DATA_BLOCK "SP201"   // DB235
// stored: MemoryReserve 100
   VAR
      "MAIN OP AUTO INITIATE PBL (GREEN)" : Bool := FALSE;
      "MAIN OP STOP PBL (RED)" : Bool := FALSE;
      RESERVE : Bool := FALSE;
      SPARE : Bool := FALSE;
      SPARE_1 : Bool := FALSE;
      SPARE_2 : Bool := FALSE;
      SPARE_3 : Bool := FALSE;
      SPARE_4 : Bool := FALSE;
      "MAIN HMI POWER TRIPPED E110CB" : Bool := TRUE;
   END_VAR
BEGIN
END_DATA_BLOCK

DATA_BLOCK "SP202"   // DB345
// stored: MemoryReserve 100
   VAR
      "AUTO INITIATE PBL LAMP (GREEN)" : Bool := FALSE;
      "STOP PBL LAMP ON (RED)" : Bool := TRUE;
      SPARE_4 : Bool := FALSE;
      "ENABLE PBL LAMP ON (BLACK)" : Bool := FALSE;
      "SAFETY RESET PBL LAMP (BLUE)" : Bool := FALSE;
      SPARE : Bool := FALSE;
      SPARE_1 : Bool := FALSE;
      SPARE_2 : Bool := FALSE;
      "TOWER LAMP 1 ON (RED)" : Bool := TRUE;
      "TOWER LAMP 2 ON (AMBER)" : Bool := FALSE;
      "TOWER LAMP 3 ON (GREEN)" : Bool := FALSE;
      "TOWER LAMP 4 ON (WHITE)" : Bool := FALSE;
      "TOWER LAMP 5 ON (BLUE)" : Bool := FALSE;
      "Buzzer On" : Bool := FALSE;
      SPARE_3 : Bool := FALSE;
      SPARE_5 : Bool := FALSE;
   END_VAR
BEGIN
END_DATA_BLOCK

DATA_BLOCK "SP203"   // DB346
// stored: MemoryReserve 100
   VAR
      "MODE SELECT AUTO" : Bool := FALSE;
      "HOME PBL (GREEN)" : Bool := FALSE;
      "SAFETY RESET PBL (BLUE)" : Bool := FALSE;
      "SCS MODE SELECT AUTO" : Bool := FALSE;
      "MODE SELECT MANUAL" : Bool := TRUE;
      "ENABLE PBL (BLACK)" : Bool := FALSE;
      "SCS MODE SELECT SETUP" : Bool := TRUE;
      "SCS MODE SELECT DISABLE" : Bool := FALSE;
   END_VAR
BEGIN
END_DATA_BLOCK

DATA_BLOCK "SP204"   // DB344
// stored: MemoryReserve 100
   VAR
      "MAIN OP EMERGENCY STOP CH.A" : Bool := TRUE;
      SPARE : Bool := FALSE;
      SPARE_1 : Bool := FALSE;
      SPARE_2 : Bool := FALSE;
      "MAIN OP EMERGENCY STOP CH.B" : Bool := FALSE;
   END_VAR
BEGIN
END_DATA_BLOCK

DATA_BLOCK "SP205"   // DB343
// stored: MemoryReserve 100
   VAR
      "PENDANT REQUIRED PL (YELLOW)" : Bool := TRUE;
      SPARE : Bool := FALSE;
      "HOME PBL LAMP ON (GREEN)" : Bool := FALSE;
      SPARE_1 : Bool := FALSE;
      SPARE_2 : Bool := FALSE;
      SPARE_3 : Bool := FALSE;
      SPARE_4 : Bool := FALSE;
      "SCS SELECT DISABLE PL (GREEN)" : Bool := TRUE;
   END_VAR
BEGIN
END_DATA_BLOCK

DATA_BLOCK "SP501"   // DB341
// stored: MemoryReserve 100
   VAR
      "CONTROL DC POWER TRIPPED E156CB" : Bool := TRUE;
      "SAFETY DC POWER TRIPPED E218CB" : Bool := TRUE;
      "CLASS 2 SMPS POWER TRIPPED E308CB" : Bool := TRUE;
      "CLASS 2 SMPS MONITORING E310PWS" : Bool := TRUE;
      "ET200ECO PN-1 POWER TRIPPED E324CB" : Bool := TRUE;
      "ET200ECO PN-2 POWER TRIPPED E328CB" : Bool := TRUE;
      "ET200ECO PN-3 POWER TRIPPED E332CB" : Bool := TRUE;
      "ET200ECO PN-4 POWER TRIPPED E336CB" : Bool := TRUE;
      "SEPA UW IONIZER TOP MAINTERNANCE DETECTION" : Bool := FALSE;
      "SEPA UW IONIZER TOP ERROR" : Bool := TRUE;
      SPARE : Bool := FALSE;
      SPARE_1 : Bool := FALSE;
      "SEPA UW IONIZER BOTTOM MAINTERNANCE DETECTION" : Bool := FALSE;
      "SEPA UW IONIZER BOTTOM ERROR" : Bool := TRUE;
      SPARE_2 : Bool := FALSE;
      SPARE_3 : Bool := FALSE;
   END_VAR
BEGIN
END_DATA_BLOCK

DATA_BLOCK "SP502"   // DB340
// stored: MemoryReserve 100
   VAR
      "CLASS2 SMPS ALARM RESET" : Bool := FALSE;
      SPARE_4 : Bool := FALSE;
      SPARE_5 : Bool := FALSE;
      SPARE_6 : Bool := FALSE;
      SPARE_7 : Bool := FALSE;
      SPARE_8 : Bool := FALSE;
      SPARE_9 : Bool := FALSE;
      SPARE_10 : Bool := FALSE;
      "SEPA UW IONIZER TOP MAINTERNANCE DETECTION" : Bool := FALSE;
      "SEPA UW IONIZER TOP DISCHARGE STOP" : Bool := FALSE;
      SPARE : Bool := FALSE;
      SPARE_1 : Bool := FALSE;
      "SEPA UW IONIZER BOTTOM MAINTERNANCE DETECTION" : Bool := FALSE;
      "SEPA UW IONIZER BOTTOM DISCHARGE STOP" : Bool := FALSE;
   END_VAR
BEGIN
END_DATA_BLOCK

DATA_BLOCK "SP506"   // DB234
// stored: MemoryReserve 100
   VAR
      "PHMI EMERGENCY STOP CH.A" : Bool := TRUE;
      "PHMI ENABLE SWITCH CH.A" : Bool := FALSE;
      SPARE : Bool := FALSE;
      SPARE_1 : Bool := FALSE;
      "PHMI EMERGENCY STOP CH.B" : Bool := FALSE;
      "PHMI ENABLE SWITCH CH.B" : Bool := FALSE;
   END_VAR
BEGIN
END_DATA_BLOCK

DATA_BLOCK "SP507"   // DB339
// stored: MemoryReserve 100
   VAR
      "UNWINDER EPCC01 INTERLOCK" : Bool := FALSE;
      "UNWINDER EPCC02 INTERLOCK" : Bool := FALSE;
      "UNWINDER EPCC03 INTERLOCK" : Bool := FALSE;
      "UNWINDER EPCC04 INTERLOCK" : Bool := FALSE;
   END_VAR
BEGIN
END_DATA_BLOCK

DATA_BLOCK "SP508"   // DB342
// stored: MemoryReserve 100
   VAR
      "ANODE ALIGN VISION BUSY (STO)" : Bool := FALSE;
      "ANODE ALIGN VISION RESULT (OK)" : Bool := TRUE;
      "STACK VISION BUSY (STO)" : Bool := FALSE;
      "STACK VISION RESULT (OK)" : Bool := FALSE;
      "CATHODE ALIGN VISION BUSY (STO)" : Bool := FALSE;
      "CATHODE ALIGN VISION RESULT (OK)" : Bool := FALSE;
   END_VAR
BEGIN
END_DATA_BLOCK

DATA_BLOCK "IdentRfHmi"   // DB213
// stored: MemoryReserve 100
   VAR
      unitIdentRf : Array[0.."NO_OF_UNITS"] of "typeEMIdentRf";
   END_VAR
BEGIN
   unitIdentRf[0].identRfEM[0..7].selectedUnit := 0;
   unitIdentRf[0].identRfEM[0..7].selectedEM := 0;
   unitIdentRf[0].identRfEM[0..7].rfReaderId := 0;
   unitIdentRf[0].identRfEM[0..7].numberOfRf := 0;
   unitIdentRf[0].identRfEM[0].rfReader[0..1].deviceName := WSTRING#'';
   unitIdentRf[0].identRfEM[1].rfReader[0..1].deviceName := WSTRING#'';
   unitIdentRf[0].identRfEM[2].rfReader[0..1].deviceName := WSTRING#'';
   unitIdentRf[0].identRfEM[3].rfReader[0..1].deviceName := WSTRING#'';
   unitIdentRf[0].identRfEM[4].rfReader[0..1].deviceName := WSTRING#'';
   unitIdentRf[0].identRfEM[5].rfReader[0..1].deviceName := WSTRING#'';
   unitIdentRf[0].identRfEM[6].rfReader[0..1].deviceName := WSTRING#'';
   unitIdentRf[0].identRfEM[7].rfReader[0..1].deviceName := WSTRING#'';
   unitIdentRf[0].identRfEM[0].rfReader[0..1].deviceType := WSTRING#'';
   unitIdentRf[0].identRfEM[1].rfReader[0..1].deviceType := WSTRING#'';
   unitIdentRf[0].identRfEM[2].rfReader[0..1].deviceType := WSTRING#'';
   unitIdentRf[0].identRfEM[3].rfReader[0..1].deviceType := WSTRING#'';
   unitIdentRf[0].identRfEM[4].rfReader[0..1].deviceType := WSTRING#'';
   unitIdentRf[0].identRfEM[5].rfReader[0..1].deviceType := WSTRING#'';
   unitIdentRf[0].identRfEM[6].rfReader[0..1].deviceType := WSTRING#'';
   unitIdentRf[0].identRfEM[7].rfReader[0..1].deviceType := WSTRING#'';
   unitIdentRf[0].identRfEM[0].rfReader[0..1].deviceId := 0;
   unitIdentRf[0].identRfEM[1].rfReader[0..1].deviceId := 0;
   unitIdentRf[0].identRfEM[2].rfReader[0..1].deviceId := 0;
   unitIdentRf[0].identRfEM[3].rfReader[0..1].deviceId := 0;
   unitIdentRf[0].identRfEM[4].rfReader[0..1].deviceId := 0;
   unitIdentRf[0].identRfEM[5].rfReader[0..1].deviceId := 0;
   unitIdentRf[0].identRfEM[6].rfReader[0..1].deviceId := 0;
   unitIdentRf[0].identRfEM[7].rfReader[0..1].deviceId := 0;
   unitIdentRf[0].identRfEM[0].rfReader[0..1].tagType := WSTRING#'';
   unitIdentRf[0].identRfEM[1].rfReader[0..1].tagType := WSTRING#'';
   unitIdentRf[0].identRfEM[2].rfReader[0..1].tagType := WSTRING#'';
   unitIdentRf[0].identRfEM[3].rfReader[0..1].tagType := WSTRING#'';
   unitIdentRf[0].identRfEM[4].rfReader[0..1].tagType := WSTRING#'';
   unitIdentRf[0].identRfEM[5].rfReader[0..1].tagType := WSTRING#'';
   unitIdentRf[0].identRfEM[6].rfReader[0..1].tagType := WSTRING#'';
   unitIdentRf[0].identRfEM[7].rfReader[0..1].tagType := WSTRING#'';
   unitIdentRf[0].identRfEM[0].rfReader[0..1].cameraMode := WSTRING#'';
   unitIdentRf[0].identRfEM[1].rfReader[0..1].cameraMode := WSTRING#'';
   unitIdentRf[0].identRfEM[2].rfReader[0..1].cameraMode := WSTRING#'';
   unitIdentRf[0].identRfEM[3].rfReader[0..1].cameraMode := WSTRING#'';
   unitIdentRf[0].identRfEM[4].rfReader[0..1].cameraMode := WSTRING#'';
   unitIdentRf[0].identRfEM[5].rfReader[0..1].cameraMode := WSTRING#'';
   unitIdentRf[0].identRfEM[6].rfReader[0..1].cameraMode := WSTRING#'';
   unitIdentRf[0].identRfEM[7].rfReader[0..1].cameraMode := WSTRING#'';
   unitIdentRf[0].identRfEM[0].rfReader[0..1].resultState := WSTRING#'';
   unitIdentRf[0].identRfEM[1].rfReader[0..1].resultState := WSTRING#'';
   unitIdentRf[0].identRfEM[2].rfReader[0..1].resultState := WSTRING#'';
   unitIdentRf[0].identRfEM[3].rfReader[0..1].resultState := WSTRING#'';
   unitIdentRf[0].identRfEM[4].rfReader[0..1].resultState := WSTRING#'';
   unitIdentRf[0].identRfEM[5].rfReader[0..1].resultState := WSTRING#'';
   unitIdentRf[0].identRfEM[6].rfReader[0..1].resultState := WSTRING#'';
   unitIdentRf[0].identRfEM[7].rfReader[0..1].resultState := WSTRING#'';
   unitIdentRf[0].identRfEM[0].rfReader[0..1].progNo := 0;
   unitIdentRf[0].identRfEM[1].rfReader[0..1].progNo := 0;
   unitIdentRf[0].identRfEM[2].rfReader[0..1].progNo := 0;
   unitIdentRf[0].identRfEM[3].rfReader[0..1].progNo := 0;
   unitIdentRf[0].identRfEM[4].rfReader[0..1].progNo := 0;
   unitIdentRf[0].identRfEM[5].rfReader[0..1].progNo := 0;
   unitIdentRf[0].identRfEM[6].rfReader[0..1].progNo := 0;
   unitIdentRf[0].identRfEM[7].rfReader[0..1].progNo := 0;
   unitIdentRf[0].identRfEM[0].rfReader[0..1].progNumberWrite := 0;
   unitIdentRf[0].identRfEM[1].rfReader[0..1].progNumberWrite := 0;
   unitIdentRf[0].identRfEM[2].rfReader[0..1].progNumberWrite := 0;
   unitIdentRf[0].identRfEM[3].rfReader[0..1].progNumberWrite := 0;
   unitIdentRf[0].identRfEM[4].rfReader[0..1].progNumberWrite := 0;
   unitIdentRf[0].identRfEM[5].rfReader[0..1].progNumberWrite := 0;
   unitIdentRf[0].identRfEM[6].rfReader[0..1].progNumberWrite := 0;
   unitIdentRf[0].identRfEM[7].rfReader[0..1].progNumberWrite := 0;
   unitIdentRf[0].identRfEM[0].rfReader[0..1].pushbutton := 16#0000;
   unitIdentRf[0].identRfEM[1].rfReader[0..1].pushbutton := 16#0000;
   unitIdentRf[0].identRfEM[2].rfReader[0..1].pushbutton := 16#0000;
   unitIdentRf[0].identRfEM[3].rfReader[0..1].pushbutton := 16#0000;
   unitIdentRf[0].identRfEM[4].rfReader[0..1].pushbutton := 16#0000;
   unitIdentRf[0].identRfEM[5].rfReader[0..1].pushbutton := 16#0000;
   unitIdentRf[0].identRfEM[6].rfReader[0..1].pushbutton := 16#0000;
   unitIdentRf[0].identRfEM[7].rfReader[0..1].pushbutton := 16#0000;
   unitIdentRf[0].identRfEM[0].rfReader[0..1].enablePushbutton := 16#0000;
   unitIdentRf[0].identRfEM[1].rfReader[0..1].enablePushbutton := 16#0000;
   unitIdentRf[0].identRfEM[2].rfReader[0..1].enablePushbutton := 16#0000;
   unitIdentRf[0].identRfEM[3].rfReader[0..1].enablePushbutton := 16#0000;
   unitIdentRf[0].identRfEM[4].rfReader[0..1].enablePushbutton := 16#0000;
   unitIdentRf[0].identRfEM[5].rfReader[0..1].enablePushbutton := 16#0000;
   unitIdentRf[0].identRfEM[6].rfReader[0..1].enablePushbutton := 16#0000;
   unitIdentRf[0].identRfEM[7].rfReader[0..1].enablePushbutton := 16#0000;
   unitIdentRf[0].identRfEM[0].rfReader[0..1].status := 16#0000;
   unitIdentRf[0].identRfEM[1].rfReader[0..1].status := 16#0000;
   unitIdentRf[0].identRfEM[2].rfReader[0..1].status := 16#0000;
   unitIdentRf[0].identRfEM[3].rfReader[0..1].status := 16#0000;
   unitIdentRf[0].identRfEM[4].rfReader[0..1].status := 16#0000;
   unitIdentRf[0].identRfEM[5].rfReader[0..1].status := 16#0000;
   unitIdentRf[0].identRfEM[6].rfReader[0..1].status := 16#0000;
   unitIdentRf[0].identRfEM[7].rfReader[0..1].status := 16#0000;
   unitIdentRf[0].identRfEM[0].rfReader[0..1].alarmCategorie := 0;
   unitIdentRf[0].identRfEM[1].rfReader[0..1].alarmCategorie := 0;
   unitIdentRf[0].identRfEM[2].rfReader[0..1].alarmCategorie := 0;
   unitIdentRf[0].identRfEM[3].rfReader[0..1].alarmCategorie := 0;
   unitIdentRf[0].identRfEM[4].rfReader[0..1].alarmCategorie := 0;
   unitIdentRf[0].identRfEM[5].rfReader[0..1].alarmCategorie := 0;
   unitIdentRf[0].identRfEM[6].rfReader[0..1].alarmCategorie := 0;
   unitIdentRf[0].identRfEM[7].rfReader[0..1].alarmCategorie := 0;
   unitIdentRf[0].identRfEM[0].rfReader[0..1].alarmNo := 0;
   unitIdentRf[0].identRfEM[1].rfReader[0..1].alarmNo := 0;
   unitIdentRf[0].identRfEM[2].rfReader[0..1].alarmNo := 0;
   unitIdentRf[0].identRfEM[3].rfReader[0..1].alarmNo := 0;
   unitIdentRf[0].identRfEM[4].rfReader[0..1].alarmNo := 0;
   unitIdentRf[0].identRfEM[5].rfReader[0..1].alarmNo := 0;
   unitIdentRf[0].identRfEM[6].rfReader[0..1].alarmNo := 0;
   unitIdentRf[0].identRfEM[7].rfReader[0..1].alarmNo := 0;
   unitIdentRf[0].identRfEM[0].rfReader[0..1].alarmCode := 16#0000_0000;
   unitIdentRf[0].identRfEM[1].rfReader[0..1].alarmCode := 16#0000_0000;
   unitIdentRf[0].identRfEM[2].rfReader[0..1].alarmCode := 16#0000_0000;
   unitIdentRf[0].identRfEM[3].rfReader[0..1].alarmCode := 16#0000_0000;
   unitIdentRf[0].identRfEM[4].rfReader[0..1].alarmCode := 16#0000_0000;
   unitIdentRf[0].identRfEM[5].rfReader[0..1].alarmCode := 16#0000_0000;
   unitIdentRf[0].identRfEM[6].rfReader[0..1].alarmCode := 16#0000_0000;
   unitIdentRf[0].identRfEM[7].rfReader[0..1].alarmCode := 16#0000_0000;
   unitIdentRf[0].identRfEM[0].rfReader[0..1].resultColor := 0;
   unitIdentRf[0].identRfEM[1].rfReader[0..1].resultColor := 0;
   unitIdentRf[0].identRfEM[2].rfReader[0..1].resultColor := 0;
   unitIdentRf[0].identRfEM[3].rfReader[0..1].resultColor := 0;
   unitIdentRf[0].identRfEM[4].rfReader[0..1].resultColor := 0;
   unitIdentRf[0].identRfEM[5].rfReader[0..1].resultColor := 0;
   unitIdentRf[0].identRfEM[6].rfReader[0..1].resultColor := 0;
   unitIdentRf[0].identRfEM[7].rfReader[0..1].resultColor := 0;
   unitIdentRf[0].identRfEM[0].rfReader[0..1].statusColorCode := 0;
   unitIdentRf[0].identRfEM[1].rfReader[0..1].statusColorCode := 0;
   unitIdentRf[0].identRfEM[2].rfReader[0..1].statusColorCode := 0;
   unitIdentRf[0].identRfEM[3].rfReader[0..1].statusColorCode := 0;
   unitIdentRf[0].identRfEM[4].rfReader[0..1].statusColorCode := 0;
   unitIdentRf[0].identRfEM[5].rfReader[0..1].statusColorCode := 0;
   unitIdentRf[0].identRfEM[6].rfReader[0..1].statusColorCode := 0;
   unitIdentRf[0].identRfEM[7].rfReader[0..1].statusColorCode := 0;
   unitIdentRf[0].identRfEM[0].rfReader[0..1].datRead1 := '';
   unitIdentRf[0].identRfEM[1].rfReader[0..1].datRead1 := '';
   unitIdentRf[0].identRfEM[2].rfReader[0..1].datRead1 := '';
   unitIdentRf[0].identRfEM[3].rfReader[0..1].datRead1 := '';
   unitIdentRf[0].identRfEM[4].rfReader[0..1].datRead1 := '';
   unitIdentRf[0].identRfEM[5].rfReader[0..1].datRead1 := '';
   unitIdentRf[0].identRfEM[6].rfReader[0..1].datRead1 := '';
   unitIdentRf[0].identRfEM[7].rfReader[0..1].datRead1 := '';
   unitIdentRf[0].identRfEM[0].rfReader[0..1].datRead2 := '';
   unitIdentRf[0].identRfEM[1].rfReader[0..1].datRead2 := '';
   unitIdentRf[0].identRfEM[2].rfReader[0..1].datRead2 := '';
   unitIdentRf[0].identRfEM[3].rfReader[0..1].datRead2 := '';
   unitIdentRf[0].identRfEM[4].rfReader[0..1].datRead2 := '';
   unitIdentRf[0].identRfEM[5].rfReader[0..1].datRead2 := '';
   unitIdentRf[0].identRfEM[6].rfReader[0..1].datRead2 := '';
   unitIdentRf[0].identRfEM[7].rfReader[0..1].datRead2 := '';
   unitIdentRf[0].identRfEM[0].rfReader[0..1].datRead3 := '';
   unitIdentRf[0].identRfEM[1].rfReader[0..1].datRead3 := '';
   unitIdentRf[0].identRfEM[2].rfReader[0..1].datRead3 := '';
   unitIdentRf[0].identRfEM[3].rfReader[0..1].datRead3 := '';
   unitIdentRf[0].identRfEM[4].rfReader[0..1].datRead3 := '';
   unitIdentRf[0].identRfEM[5].rfReader[0..1].datRead3 := '';
   unitIdentRf[0].identRfEM[6].rfReader[0..1].datRead3 := '';
   unitIdentRf[0].identRfEM[7].rfReader[0..1].datRead3 := '';
   unitIdentRf[0].identRfEM[0].rfReader[0..1].datRead4 := '';
   unitIdentRf[0].identRfEM[1].rfReader[0..1].datRead4 := '';
   unitIdentRf[0].identRfEM[2].rfReader[0..1].datRead4 := '';
   unitIdentRf[0].identRfEM[3].rfReader[0..1].datRead4 := '';
   unitIdentRf[0].identRfEM[4].rfReader[0..1].datRead4 := '';
   unitIdentRf[0].identRfEM[5].rfReader[0..1].datRead4 := '';
   unitIdentRf[0].identRfEM[6].rfReader[0..1].datRead4 := '';
   unitIdentRf[0].identRfEM[7].rfReader[0..1].datRead4 := '';
   unitIdentRf[0].identRfEM[0].rfReader[0..1].datWrite1 := '';
   unitIdentRf[0].identRfEM[1].rfReader[0..1].datWrite1 := '';
   unitIdentRf[0].identRfEM[2].rfReader[0..1].datWrite1 := '';
   unitIdentRf[0].identRfEM[3].rfReader[0..1].datWrite1 := '';
   unitIdentRf[0].identRfEM[4].rfReader[0..1].datWrite1 := '';
   unitIdentRf[0].identRfEM[5].rfReader[0..1].datWrite1 := '';
   unitIdentRf[0].identRfEM[6].rfReader[0..1].datWrite1 := '';
   unitIdentRf[0].identRfEM[7].rfReader[0..1].datWrite1 := '';
   unitIdentRf[0].identRfEM[0].rfReader[0..1].datWrite2 := '';
   unitIdentRf[0].identRfEM[1].rfReader[0..1].datWrite2 := '';
   unitIdentRf[0].identRfEM[2].rfReader[0..1].datWrite2 := '';
   unitIdentRf[0].identRfEM[3].rfReader[0..1].datWrite2 := '';
   unitIdentRf[0].identRfEM[4].rfReader[0..1].datWrite2 := '';
   unitIdentRf[0].identRfEM[5].rfReader[0..1].datWrite2 := '';
   unitIdentRf[0].identRfEM[6].rfReader[0..1].datWrite2 := '';
   unitIdentRf[0].identRfEM[7].rfReader[0..1].datWrite2 := '';
   unitIdentRf[0].identRfEM[0].rfReader[0..1].datWrite3 := '';
   unitIdentRf[0].identRfEM[1].rfReader[0..1].datWrite3 := '';
   unitIdentRf[0].identRfEM[2].rfReader[0..1].datWrite3 := '';
   unitIdentRf[0].identRfEM[3].rfReader[0..1].datWrite3 := '';
   unitIdentRf[0].identRfEM[4].rfReader[0..1].datWrite3 := '';
   unitIdentRf[0].identRfEM[5].rfReader[0..1].datWrite3 := '';
   unitIdentRf[0].identRfEM[6].rfReader[0..1].datWrite3 := '';
   unitIdentRf[0].identRfEM[7].rfReader[0..1].datWrite3 := '';
   unitIdentRf[0].identRfEM[0].rfReader[0..1].datWrite4 := '';
   unitIdentRf[0].identRfEM[1].rfReader[0..1].datWrite4 := '';
   unitIdentRf[0].identRfEM[2].rfReader[0..1].datWrite4 := '';
   unitIdentRf[0].identRfEM[3].rfReader[0..1].datWrite4 := '';
   unitIdentRf[0].identRfEM[4].rfReader[0..1].datWrite4 := '';
   unitIdentRf[0].identRfEM[5].rfReader[0..1].datWrite4 := '';
   unitIdentRf[0].identRfEM[6].rfReader[0..1].datWrite4 := '';
   unitIdentRf[0].identRfEM[7].rfReader[0..1].datWrite4 := '';
END_DATA_BLOCK

DATA_BLOCK "IdentMvHmi"   // DB214
// stored: MemoryReserve 100
   VAR
      unitIdentMv : Array[0.."NO_OF_UNITS"] of "typeEMIdentMv";
   END_VAR
BEGIN
   unitIdentMv[0].identMvEM[0..7].selectedUnit := 0;
   unitIdentMv[0].identMvEM[0..7].selectedEM := 0;
   unitIdentMv[0].identMvEM[0..7].mvReaderId := 0;
   unitIdentMv[0].identMvEM[0..7].numberOfMv := 0;
   unitIdentMv[0].identMvEM[0].mvReader[0..1].deviceName := WSTRING#'';
   unitIdentMv[0].identMvEM[1].mvReader[0..1].deviceName := WSTRING#'';
   unitIdentMv[0].identMvEM[2].mvReader[0..1].deviceName := WSTRING#'';
   unitIdentMv[0].identMvEM[3].mvReader[0..1].deviceName := WSTRING#'';
   unitIdentMv[0].identMvEM[4].mvReader[0..1].deviceName := WSTRING#'';
   unitIdentMv[0].identMvEM[5].mvReader[0..1].deviceName := WSTRING#'';
   unitIdentMv[0].identMvEM[6].mvReader[0..1].deviceName := WSTRING#'';
   unitIdentMv[0].identMvEM[7].mvReader[0..1].deviceName := WSTRING#'';
   unitIdentMv[0].identMvEM[0].mvReader[0..1].deviceType := WSTRING#'';
   unitIdentMv[0].identMvEM[1].mvReader[0..1].deviceType := WSTRING#'';
   unitIdentMv[0].identMvEM[2].mvReader[0..1].deviceType := WSTRING#'';
   unitIdentMv[0].identMvEM[3].mvReader[0..1].deviceType := WSTRING#'';
   unitIdentMv[0].identMvEM[4].mvReader[0..1].deviceType := WSTRING#'';
   unitIdentMv[0].identMvEM[5].mvReader[0..1].deviceType := WSTRING#'';
   unitIdentMv[0].identMvEM[6].mvReader[0..1].deviceType := WSTRING#'';
   unitIdentMv[0].identMvEM[7].mvReader[0..1].deviceType := WSTRING#'';
   unitIdentMv[0].identMvEM[0].mvReader[0..1].deviceId := 0;
   unitIdentMv[0].identMvEM[1].mvReader[0..1].deviceId := 0;
   unitIdentMv[0].identMvEM[2].mvReader[0..1].deviceId := 0;
   unitIdentMv[0].identMvEM[3].mvReader[0..1].deviceId := 0;
   unitIdentMv[0].identMvEM[4].mvReader[0..1].deviceId := 0;
   unitIdentMv[0].identMvEM[5].mvReader[0..1].deviceId := 0;
   unitIdentMv[0].identMvEM[6].mvReader[0..1].deviceId := 0;
   unitIdentMv[0].identMvEM[7].mvReader[0..1].deviceId := 0;
   unitIdentMv[0].identMvEM[0].mvReader[0..1].tagType := WSTRING#'';
   unitIdentMv[0].identMvEM[1].mvReader[0..1].tagType := WSTRING#'';
   unitIdentMv[0].identMvEM[2].mvReader[0..1].tagType := WSTRING#'';
   unitIdentMv[0].identMvEM[3].mvReader[0..1].tagType := WSTRING#'';
   unitIdentMv[0].identMvEM[4].mvReader[0..1].tagType := WSTRING#'';
   unitIdentMv[0].identMvEM[5].mvReader[0..1].tagType := WSTRING#'';
   unitIdentMv[0].identMvEM[6].mvReader[0..1].tagType := WSTRING#'';
   unitIdentMv[0].identMvEM[7].mvReader[0..1].tagType := WSTRING#'';
   unitIdentMv[0].identMvEM[0].mvReader[0..1].cameraMode := WSTRING#'';
   unitIdentMv[0].identMvEM[1].mvReader[0..1].cameraMode := WSTRING#'';
   unitIdentMv[0].identMvEM[2].mvReader[0..1].cameraMode := WSTRING#'';
   unitIdentMv[0].identMvEM[3].mvReader[0..1].cameraMode := WSTRING#'';
   unitIdentMv[0].identMvEM[4].mvReader[0..1].cameraMode := WSTRING#'';
   unitIdentMv[0].identMvEM[5].mvReader[0..1].cameraMode := WSTRING#'';
   unitIdentMv[0].identMvEM[6].mvReader[0..1].cameraMode := WSTRING#'';
   unitIdentMv[0].identMvEM[7].mvReader[0..1].cameraMode := WSTRING#'';
   unitIdentMv[0].identMvEM[0].mvReader[0..1].resultState := WSTRING#'';
   unitIdentMv[0].identMvEM[1].mvReader[0..1].resultState := WSTRING#'';
   unitIdentMv[0].identMvEM[2].mvReader[0..1].resultState := WSTRING#'';
   unitIdentMv[0].identMvEM[3].mvReader[0..1].resultState := WSTRING#'';
   unitIdentMv[0].identMvEM[4].mvReader[0..1].resultState := WSTRING#'';
   unitIdentMv[0].identMvEM[5].mvReader[0..1].resultState := WSTRING#'';
   unitIdentMv[0].identMvEM[6].mvReader[0..1].resultState := WSTRING#'';
   unitIdentMv[0].identMvEM[7].mvReader[0..1].resultState := WSTRING#'';
   unitIdentMv[0].identMvEM[0].mvReader[0..1].progNo := 0;
   unitIdentMv[0].identMvEM[1].mvReader[0..1].progNo := 0;
   unitIdentMv[0].identMvEM[2].mvReader[0..1].progNo := 0;
   unitIdentMv[0].identMvEM[3].mvReader[0..1].progNo := 0;
   unitIdentMv[0].identMvEM[4].mvReader[0..1].progNo := 0;
   unitIdentMv[0].identMvEM[5].mvReader[0..1].progNo := 0;
   unitIdentMv[0].identMvEM[6].mvReader[0..1].progNo := 0;
   unitIdentMv[0].identMvEM[7].mvReader[0..1].progNo := 0;
   unitIdentMv[0].identMvEM[0].mvReader[0..1].progNumberWrite := 0;
   unitIdentMv[0].identMvEM[1].mvReader[0..1].progNumberWrite := 0;
   unitIdentMv[0].identMvEM[2].mvReader[0..1].progNumberWrite := 0;
   unitIdentMv[0].identMvEM[3].mvReader[0..1].progNumberWrite := 0;
   unitIdentMv[0].identMvEM[4].mvReader[0..1].progNumberWrite := 0;
   unitIdentMv[0].identMvEM[5].mvReader[0..1].progNumberWrite := 0;
   unitIdentMv[0].identMvEM[6].mvReader[0..1].progNumberWrite := 0;
   unitIdentMv[0].identMvEM[7].mvReader[0..1].progNumberWrite := 0;
   unitIdentMv[0].identMvEM[0].mvReader[0..1].pushbutton := 16#0000;
   unitIdentMv[0].identMvEM[1].mvReader[0..1].pushbutton := 16#0000;
   unitIdentMv[0].identMvEM[2].mvReader[0..1].pushbutton := 16#0000;
   unitIdentMv[0].identMvEM[3].mvReader[0..1].pushbutton := 16#0000;
   unitIdentMv[0].identMvEM[4].mvReader[0..1].pushbutton := 16#0000;
   unitIdentMv[0].identMvEM[5].mvReader[0..1].pushbutton := 16#0000;
   unitIdentMv[0].identMvEM[6].mvReader[0..1].pushbutton := 16#0000;
   unitIdentMv[0].identMvEM[7].mvReader[0..1].pushbutton := 16#0000;
   unitIdentMv[0].identMvEM[0].mvReader[0..1].enablePushbutton := 16#0000;
   unitIdentMv[0].identMvEM[1].mvReader[0..1].enablePushbutton := 16#0000;
   unitIdentMv[0].identMvEM[2].mvReader[0..1].enablePushbutton := 16#0000;
   unitIdentMv[0].identMvEM[3].mvReader[0..1].enablePushbutton := 16#0000;
   unitIdentMv[0].identMvEM[4].mvReader[0..1].enablePushbutton := 16#0000;
   unitIdentMv[0].identMvEM[5].mvReader[0..1].enablePushbutton := 16#0000;
   unitIdentMv[0].identMvEM[6].mvReader[0..1].enablePushbutton := 16#0000;
   unitIdentMv[0].identMvEM[7].mvReader[0..1].enablePushbutton := 16#0000;
   unitIdentMv[0].identMvEM[0].mvReader[0..1].status := 16#0000;
   unitIdentMv[0].identMvEM[1].mvReader[0..1].status := 16#0000;
   unitIdentMv[0].identMvEM[2].mvReader[0..1].status := 16#0000;
   unitIdentMv[0].identMvEM[3].mvReader[0..1].status := 16#0000;
   unitIdentMv[0].identMvEM[4].mvReader[0..1].status := 16#0000;
   unitIdentMv[0].identMvEM[5].mvReader[0..1].status := 16#0000;
   unitIdentMv[0].identMvEM[6].mvReader[0..1].status := 16#0000;
   unitIdentMv[0].identMvEM[7].mvReader[0..1].status := 16#0000;
   unitIdentMv[0].identMvEM[0].mvReader[0..1].alarmCategorie := 0;
   unitIdentMv[0].identMvEM[1].mvReader[0..1].alarmCategorie := 0;
   unitIdentMv[0].identMvEM[2].mvReader[0..1].alarmCategorie := 0;
   unitIdentMv[0].identMvEM[3].mvReader[0..1].alarmCategorie := 0;
   unitIdentMv[0].identMvEM[4].mvReader[0..1].alarmCategorie := 0;
   unitIdentMv[0].identMvEM[5].mvReader[0..1].alarmCategorie := 0;
   unitIdentMv[0].identMvEM[6].mvReader[0..1].alarmCategorie := 0;
   unitIdentMv[0].identMvEM[7].mvReader[0..1].alarmCategorie := 0;
   unitIdentMv[0].identMvEM[0].mvReader[0..1].alarmNo := 0;
   unitIdentMv[0].identMvEM[1].mvReader[0..1].alarmNo := 0;
   unitIdentMv[0].identMvEM[2].mvReader[0..1].alarmNo := 0;
   unitIdentMv[0].identMvEM[3].mvReader[0..1].alarmNo := 0;
   unitIdentMv[0].identMvEM[4].mvReader[0..1].alarmNo := 0;
   unitIdentMv[0].identMvEM[5].mvReader[0..1].alarmNo := 0;
   unitIdentMv[0].identMvEM[6].mvReader[0..1].alarmNo := 0;
   unitIdentMv[0].identMvEM[7].mvReader[0..1].alarmNo := 0;
   unitIdentMv[0].identMvEM[0].mvReader[0..1].alarmCode := 16#0000_0000;
   unitIdentMv[0].identMvEM[1].mvReader[0..1].alarmCode := 16#0000_0000;
   unitIdentMv[0].identMvEM[2].mvReader[0..1].alarmCode := 16#0000_0000;
   unitIdentMv[0].identMvEM[3].mvReader[0..1].alarmCode := 16#0000_0000;
   unitIdentMv[0].identMvEM[4].mvReader[0..1].alarmCode := 16#0000_0000;
   unitIdentMv[0].identMvEM[5].mvReader[0..1].alarmCode := 16#0000_0000;
   unitIdentMv[0].identMvEM[6].mvReader[0..1].alarmCode := 16#0000_0000;
   unitIdentMv[0].identMvEM[7].mvReader[0..1].alarmCode := 16#0000_0000;
   unitIdentMv[0].identMvEM[0].mvReader[0..1].resultColor := 0;
   unitIdentMv[0].identMvEM[1].mvReader[0..1].resultColor := 0;
   unitIdentMv[0].identMvEM[2].mvReader[0..1].resultColor := 0;
   unitIdentMv[0].identMvEM[3].mvReader[0..1].resultColor := 0;
   unitIdentMv[0].identMvEM[4].mvReader[0..1].resultColor := 0;
   unitIdentMv[0].identMvEM[5].mvReader[0..1].resultColor := 0;
   unitIdentMv[0].identMvEM[6].mvReader[0..1].resultColor := 0;
   unitIdentMv[0].identMvEM[7].mvReader[0..1].resultColor := 0;
   unitIdentMv[0].identMvEM[0].mvReader[0..1].statusColorCode := 0;
   unitIdentMv[0].identMvEM[1].mvReader[0..1].statusColorCode := 0;
   unitIdentMv[0].identMvEM[2].mvReader[0..1].statusColorCode := 0;
   unitIdentMv[0].identMvEM[3].mvReader[0..1].statusColorCode := 0;
   unitIdentMv[0].identMvEM[4].mvReader[0..1].statusColorCode := 0;
   unitIdentMv[0].identMvEM[5].mvReader[0..1].statusColorCode := 0;
   unitIdentMv[0].identMvEM[6].mvReader[0..1].statusColorCode := 0;
   unitIdentMv[0].identMvEM[7].mvReader[0..1].statusColorCode := 0;
   unitIdentMv[0].identMvEM[0].mvReader[0..1].datRead1 := '';
   unitIdentMv[0].identMvEM[1].mvReader[0..1].datRead1 := '';
   unitIdentMv[0].identMvEM[2].mvReader[0..1].datRead1 := '';
   unitIdentMv[0].identMvEM[3].mvReader[0..1].datRead1 := '';
   unitIdentMv[0].identMvEM[4].mvReader[0..1].datRead1 := '';
   unitIdentMv[0].identMvEM[5].mvReader[0..1].datRead1 := '';
   unitIdentMv[0].identMvEM[6].mvReader[0..1].datRead1 := '';
   unitIdentMv[0].identMvEM[7].mvReader[0..1].datRead1 := '';
   unitIdentMv[0].identMvEM[0].mvReader[0..1].datRead2 := '';
   unitIdentMv[0].identMvEM[1].mvReader[0..1].datRead2 := '';
   unitIdentMv[0].identMvEM[2].mvReader[0..1].datRead2 := '';
   unitIdentMv[0].identMvEM[3].mvReader[0..1].datRead2 := '';
   unitIdentMv[0].identMvEM[4].mvReader[0..1].datRead2 := '';
   unitIdentMv[0].identMvEM[5].mvReader[0..1].datRead2 := '';
   unitIdentMv[0].identMvEM[6].mvReader[0..1].datRead2 := '';
   unitIdentMv[0].identMvEM[7].mvReader[0..1].datRead2 := '';
   unitIdentMv[0].identMvEM[0].mvReader[0..1].datRead3 := '';
   unitIdentMv[0].identMvEM[1].mvReader[0..1].datRead3 := '';
   unitIdentMv[0].identMvEM[2].mvReader[0..1].datRead3 := '';
   unitIdentMv[0].identMvEM[3].mvReader[0..1].datRead3 := '';
   unitIdentMv[0].identMvEM[4].mvReader[0..1].datRead3 := '';
   unitIdentMv[0].identMvEM[5].mvReader[0..1].datRead3 := '';
   unitIdentMv[0].identMvEM[6].mvReader[0..1].datRead3 := '';
   unitIdentMv[0].identMvEM[7].mvReader[0..1].datRead3 := '';
   unitIdentMv[0].identMvEM[0].mvReader[0..1].datRead4 := '';
   unitIdentMv[0].identMvEM[1].mvReader[0..1].datRead4 := '';
   unitIdentMv[0].identMvEM[2].mvReader[0..1].datRead4 := '';
   unitIdentMv[0].identMvEM[3].mvReader[0..1].datRead4 := '';
   unitIdentMv[0].identMvEM[4].mvReader[0..1].datRead4 := '';
   unitIdentMv[0].identMvEM[5].mvReader[0..1].datRead4 := '';
   unitIdentMv[0].identMvEM[6].mvReader[0..1].datRead4 := '';
   unitIdentMv[0].identMvEM[7].mvReader[0..1].datRead4 := '';
   unitIdentMv[0].identMvEM[0].mvReader[0].datWrite1 := '';
   unitIdentMv[0].identMvEM[0].mvReader[1].datWrite1 := 'Siemens';
   unitIdentMv[0].identMvEM[1].mvReader[0..1].datWrite1 := '';
   unitIdentMv[0].identMvEM[2].mvReader[0..1].datWrite1 := '';
   unitIdentMv[0].identMvEM[3].mvReader[0..1].datWrite1 := '';
   unitIdentMv[0].identMvEM[4].mvReader[0..1].datWrite1 := '';
   unitIdentMv[0].identMvEM[5].mvReader[0..1].datWrite1 := '';
   unitIdentMv[0].identMvEM[6].mvReader[0..1].datWrite1 := '';
   unitIdentMv[0].identMvEM[7].mvReader[0..1].datWrite1 := '';
   unitIdentMv[0].identMvEM[0].mvReader[0..1].datWrite2 := '';
   unitIdentMv[0].identMvEM[1].mvReader[0..1].datWrite2 := '';
   unitIdentMv[0].identMvEM[2].mvReader[0..1].datWrite2 := '';
   unitIdentMv[0].identMvEM[3].mvReader[0..1].datWrite2 := '';
   unitIdentMv[0].identMvEM[4].mvReader[0..1].datWrite2 := '';
   unitIdentMv[0].identMvEM[5].mvReader[0..1].datWrite2 := '';
   unitIdentMv[0].identMvEM[6].mvReader[0..1].datWrite2 := '';
   unitIdentMv[0].identMvEM[7].mvReader[0..1].datWrite2 := '';
   unitIdentMv[0].identMvEM[0].mvReader[0..1].datWrite3 := '';
   unitIdentMv[0].identMvEM[1].mvReader[0..1].datWrite3 := '';
   unitIdentMv[0].identMvEM[2].mvReader[0..1].datWrite3 := '';
   unitIdentMv[0].identMvEM[3].mvReader[0..1].datWrite3 := '';
   unitIdentMv[0].identMvEM[4].mvReader[0..1].datWrite3 := '';
   unitIdentMv[0].identMvEM[5].mvReader[0..1].datWrite3 := '';
   unitIdentMv[0].identMvEM[6].mvReader[0..1].datWrite3 := '';
   unitIdentMv[0].identMvEM[7].mvReader[0..1].datWrite3 := '';
   unitIdentMv[0].identMvEM[0].mvReader[0..1].datWrite4 := '';
   unitIdentMv[0].identMvEM[1].mvReader[0..1].datWrite4 := '';
   unitIdentMv[0].identMvEM[2].mvReader[0..1].datWrite4 := '';
   unitIdentMv[0].identMvEM[3].mvReader[0..1].datWrite4 := '';
   unitIdentMv[0].identMvEM[4].mvReader[0..1].datWrite4 := '';
   unitIdentMv[0].identMvEM[5].mvReader[0..1].datWrite4 := '';
   unitIdentMv[0].identMvEM[6].mvReader[0..1].datWrite4 := '';
   unitIdentMv[0].identMvEM[7].mvReader[0..1].datWrite4 := '';
END_DATA_BLOCK

DATA_BLOCK "BK01"   // DB87
// stored: MemoryReserve 100
   VAR
      "X10-1.BTM DIRECTION CHECK SENSOR" : Bool := TRUE;
      "X11-1.SEPA UNWINDER IONIZER TOP 2 POWER" : Bool := FALSE;
      "X12-1.SPARE" : Bool := FALSE;
      "X13-1.COMPENSATOR #1 LIMIT SENSOR(-)" : Bool := TRUE;
      "X14-1.COMPENSATOR #1 LIMIT SENSOR(+)" : Bool := TRUE;
      "X15-1.SPARE" : Bool := FALSE;
      "X16-1.SPARE" : Bool := FALSE;
      "X17-1.SAFETY PIN IDLE POSITION" : Bool := TRUE;
      "X10-2.TOP DIRECTION CHECK SENSOR" : Bool := FALSE;
      "X11-2.SEPA UNWINDER IONIZER BTM 2 POWER" : Bool := FALSE;
      "X12-2.SPARE" : Bool := FALSE;
      "X13-2.COMPENSATOR #1 HOME SENSOR" : Bool := TRUE;
      "X14-2.SPARE" : Bool := FALSE;
      "X15-2.SPARE" : Bool := FALSE;
      "X16-2.SPARE" : Bool := FALSE;
      "X17-2.SPARE" : Bool := FALSE;
   END_VAR
BEGIN
END_DATA_BLOCK

DATA_BLOCK "BK02"   // DB304
// stored: MemoryReserve 100
   VAR
      "X10-1.SUCTION PAD TOP DOWN" : Bool := TRUE;
      "X11-1.SUCTION PAD BTM DOWN" : Bool := TRUE;
      "X12-1.CUTTER DOWN" : Bool := TRUE;
      "X13-1.TAPE TOP DOWN" : Bool := FALSE;
      "X14-1.TAPE BTM DOWN" : Bool := TRUE;
      "X15-1.SPLICE HEAD ROTATE TOP BACKWARD" : Bool := TRUE;
      "X16-1.SPLICE HEAD ROTATE BTM BACKWARD" : Bool := TRUE;
      "X17-1.SPARE" : Bool := FALSE;
      "X10-2.SUCTION PAD TOP UP" : Bool := FALSE;
      "X11-2.SUCTION PAD BTM UP" : Bool := FALSE;
      "X12-2.CUTTER UP" : Bool := FALSE;
      "X13-2.TAPE TOP UP" : Bool := TRUE;
      "X14-2.TAPE BTM UP" : Bool := FALSE;
      "X15-2.SPLICE HEAD ROTATE TOP FORWARD" : Bool := FALSE;
      "X16-2.SPLICE HEAD ROTATE BTM FORWARD" : Bool := FALSE;
      "X17-2.SPARE" : Bool := FALSE;
   END_VAR
BEGIN
END_DATA_BLOCK

DATA_BLOCK "BK03"   // DB316
// stored: MemoryReserve 100
   VAR
      "X10-1.SUCTION PAD TOP LEFT PRESSURE SWITCH" : Bool := FALSE;
      "X10-2.SUCTION PAD TOP RIGHT PRESSURE SWITCH" : Bool := FALSE;
      "X12-1.SUCTION PAD BTM LEFT PRESSURE SWITCH" : Bool := FALSE;
      "X12-2.SUCTION PAD BTM RIGHT PRESSURE SWITCH" : Bool := FALSE;
      "X14-1.SUCTION PAD TOP TAPE PRESSURE SWITCH" : Bool := FALSE;
      "X14-2.SUCTION PAD BTM TAPE PRESSURE SWITCH" : Bool := FALSE;
      "X16-1.ROTATION SAFETY PIN POSITION" : Bool := FALSE;
      "X16-2.SPARE" : Bool := FALSE;
   END_VAR
BEGIN
END_DATA_BLOCK

DATA_BLOCK "BK04"   // DB308
// stored: MemoryReserve 100
   VAR
      "X10-1.CATHODE MAIN P&P1 LIMITS SENSOR(-)" : Bool := TRUE;
      "X11-1.CATHODE MAIN P&P1 LIMITS SENSOR(+)" : Bool := TRUE;
      "X12-1.CATHODE MAIN P&P2 LIMITS SENSOR(-)" : Bool := TRUE;
      "X13-1.CATHODE MAIN P&P2 LIMITS SENSOR(+)" : Bool := TRUE;
      "X14-1.ANODE MAIN P&P2 LIMITS SENSOR(-)" : Bool := TRUE;
      "X15-1.ANODE MAIN P&P2 LIMITS SENSOR(+)" : Bool := TRUE;
      "X16-1.ANODE MAIN P&P1 LIMITS SENSOR(-)" : Bool := TRUE;
      "X17-1.ANODE MAIN P&P1 LIMITS SENSOR(+)" : Bool := TRUE;
      "X10-2.CATHODE MAIN P&P1 LIMITS SENSOR HOME" : Bool := TRUE;
      "X11-2.SPARE" : Bool := FALSE;
      "X12-2.CATHODE MAIN P&P2 LIMITS SENSOR HOME" : Bool := TRUE;
      "X13-2.SPARE" : Bool := FALSE;
      "X14-2.ANODE MAIN P&P2 LIMITS SENSOR HOME" : Bool := TRUE;
      "X15-2.SPARE" : Bool := FALSE;
      "X16-2.ANODE MAIN P&P1 LIMITS SENSOR HOME" : Bool := TRUE;
      "X17-2.SPARE" : Bool := FALSE;
   END_VAR
BEGIN
END_DATA_BLOCK

DATA_BLOCK "BK05"   // DB307
// stored: MemoryReserve 100
   VAR
      "X10-1.ANODE MAIN P&P1 Z-AXIS LIMIT SENSOR(-)" : Bool := TRUE;
      "X11-1.ANODE MAIN P&P1 Z-AXIS LIMIT SENSOR(+)" : Bool := TRUE;
      "X12-1.ANODE MAIN P&P1 Y-AXIS LIMIT SENSOR(-)" : Bool := TRUE;
      "X13-1.ANODE MAIN P&P1 Y-AXIS LIMIT SENSOR(+)" : Bool := TRUE;
      "X14-1.SPARE" : Bool := FALSE;
      "X15-1.ANODE MAIN P&P1 DETECT SENSOR" : Bool := FALSE;
      "X16-1.ANODE MAIN P&P1 ROTARY CCW" : Bool := FALSE;
      "X17-1.ANODE MAIN P&P1 PRESSURE SWITCH" : Bool := FALSE;
      "X10-2.ANODE MAIN P&P1 Z-AXIS HOME SENSOR" : Bool := TRUE;
      "X11-2.SPARE" : Bool := FALSE;
      "X12-2.ANODE MAIN P&P1 Y-AXIS HOME SENSOR" : Bool := TRUE;
      "X13-2.SPARE" : Bool := FALSE;
      "X14-2.SPARE" : Bool := FALSE;
      "X15-2.SPARE" : Bool := FALSE;
      "X16-2.ANODE MAIN P&P1 ROTARY CW" : Bool := TRUE;
      "X17-2.SPARE" : Bool := FALSE;
   END_VAR
BEGIN
END_DATA_BLOCK

DATA_BLOCK "BK06"   // DB310
// stored: MemoryReserve 100
   VAR
      "X10-1.ANODE MAIN P&P2 Z-AXIS LIMIT SENSOR(-)" : Bool := TRUE;
      "X10-2.ANODE MAIN P&P2 Z-AXIS HOME SENSOR" : Bool := TRUE;
      "X12-1.ANODE MAIN P&P2 Z-AXIS LIMIT SENSOR(+)" : Bool := TRUE;
      "X12-2.ANODE MAIN P&P2 DETECT SENSOR" : Bool := FALSE;
      "X14-1.ANODE MAIN P&P2 PRESSURE SWITCH" : Bool := FALSE;
      "X14-2.SPARE" : Bool := FALSE;
      "X16-1.SPARE" : Bool := FALSE;
      "X16-2.SPARE" : Bool := FALSE;
   END_VAR
BEGIN
END_DATA_BLOCK

DATA_BLOCK "BK07"   // DB303
// stored: MemoryReserve 100
   VAR
      "X10-1.CATHODE MAIN P&P1 Z-AXIS LIMIT SENSOR(-)" : Bool := TRUE;
      "X11-1.CATHODE MAIN P&P1 Z-AXIS LIMIT SENSOR(+)" : Bool := TRUE;
      "X12-1.CATHODE MAIN P&P1 Y-AXIS LIMIT SENSOR(-)" : Bool := TRUE;
      "X13-1.CATHODE MAIN P&P1 Y-AXIS LIMIT SENSOR(+)" : Bool := TRUE;
      "X14-1.SPARE" : Bool := FALSE;
      "X15-1.CATHODE MAIN P&P1 DETECT SENSOR" : Bool := FALSE;
      "X16-1.CATHODE MAIN P&P1 ROTARY CCW" : Bool := FALSE;
      "X17-1.CATHODE MAIN P&P1 PRESSURE SWITCH" : Bool := FALSE;
      "X10-2.CATHODE MAIN P&P1 Z-AXIS HOME SENSOR" : Bool := TRUE;
      "X11-2.SPARE" : Bool := FALSE;
      "X12-2.CATHODE MAIN P&P1 Y-AXIS HOME SENSOR" : Bool := TRUE;
      "X13-2.SPARE" : Bool := FALSE;
      "X14-2.SPARE" : Bool := FALSE;
      "X15-2.SPARE" : Bool := FALSE;
      "X16-2.CATHODE MAIN P&P1 ROTARY CW" : Bool := FALSE;
      "X17-2.SPARE" : Bool := FALSE;
   END_VAR
BEGIN
END_DATA_BLOCK

DATA_BLOCK "BK08"   // DB315
// stored: MemoryReserve 100
   VAR
      "X10-1.CATHODE MAIN P&P2 Z-AXIS LIMIT SENSOR(-)" : Bool := TRUE;
      "X10-2.CATHODE MAIN P&P2 Z-AXIS HOME SENSOR" : Bool := TRUE;
      "X12-1.CATHODE MAIN P&P2 Z-AXIS LIMIT SENSOR(+)" : Bool := TRUE;
      "X12-2.CATHODE MAIN P&P2 DETECT SENSOR" : Bool := FALSE;
      "X14-1.CATHODE MAIN P&P2 PRESSURE SWITCH" : Bool := FALSE;
      "X14-2.SPARE" : Bool := FALSE;
      "X16-1.SPARE" : Bool := FALSE;
      "X16-2.SPARE" : Bool := FALSE;
   END_VAR
BEGIN
END_DATA_BLOCK

DATA_BLOCK "BK09"   // DB302
// stored: MemoryReserve 100
   VAR
      "X10-1.ANODE ALIGN TABLE Y2-AXIS LIMIT SENSOR(-)" : Bool := TRUE;
      "X11-1.ANODE ALIGN TABLE Y2-AXIS LIMIT SENSOR(+)" : Bool := TRUE;
      "X12-1.ANODE ALIGN TABLE X-AXIS LIMIT SENSOR(-)" : Bool := TRUE;
      "X13-1.ANODE ALIGN TABLE X-AXIS LIMIT SENSOR(+)" : Bool := TRUE;
      "X14-1.ANODE ALIGN TABLE Y1-AXIS LIMIT SENSOR(-)" : Bool := TRUE;
      "X15-1.ANODE ALIGN TABLE Y1-AXIS LIMIT SENSOR(+)" : Bool := TRUE;
      "X16-1.ANODE ALIGN TABLE ELECTRODE DETECT SENSOR" : Bool := FALSE;
      "X17-1.ANODE ALIGN TABLE PRESSURE SWITCH" : Bool := FALSE;
      "X10-2.ANODE ALIGN TABLE Y2-AXIS HOME SENSOR" : Bool := TRUE;
      "X11-2.SPARE" : Bool := FALSE;
      "X12-2.ANODE ALIGN TABLE X-AXIS HOME SENSOR" : Bool := FALSE;
      "X13-2.SPARE" : Bool := FALSE;
      "X14-2.ANODE ALIGN TABLE Y1-AXIS HOME SENSOR" : Bool := TRUE;
      "X15-2.SPARE" : Bool := FALSE;
      "X16-2.SPARE" : Bool := FALSE;
      "X17-2.SPARE" : Bool := FALSE;
   END_VAR
BEGIN
END_DATA_BLOCK

DATA_BLOCK "BK10"   // DB306
// stored: MemoryReserve 100
   VAR
      "X10-1.ANODE FIX FRONT BACKWARD" : Bool := TRUE;
      "X11-1.SEPA CLAMP SAFETY PIN DETECT SENSOR" : Bool := FALSE;
      "X12-1.ANODE FIX REAR BACKWARD" : Bool := TRUE;
      "X13-1.SEPA CLAMP PRESSURE SWITCH" : Bool := FALSE;
      "X14-1.FIX ANODE DETECT SENSOR" : Bool := FALSE;
      "X15-1.SPARE" : Bool := FALSE;
      "X16-1.SPARE" : Bool := FALSE;
      "X17-1.SPARE" : Bool := FALSE;
      "X10-2.ANODE FIX FRONT FORWARD" : Bool := FALSE;
      "X11-2.SEPA GRIPPER SAFETY PIN DETECT SENSOR" : Bool := FALSE;
      "X12-2.ANODE FIX REAR FORWARD" : Bool := FALSE;
      "X13-2.SPARE" : Bool := FALSE;
      "X14-2.SPARE" : Bool := FALSE;
      "X15-2.SPARE" : Bool := FALSE;
      "X16-2.SPARE" : Bool := FALSE;
      "X17-2.SPARE" : Bool := FALSE;
   END_VAR
BEGIN
END_DATA_BLOCK

DATA_BLOCK "BK11"   // DB305
// stored: MemoryReserve 100
   VAR
      "X10-1.ANODE NG BOX FULL SENSOR" : Bool := TRUE;
      "X10-2.SPARE" : Bool := FALSE;
      "X12-1.ANODE NG BOX LIFT DOWN" : Bool := FALSE;
      "X12-2.ANODE NG BOX LIFT UP" : Bool := TRUE;
      "X14-1.ANODE NG BOX LOCK DOWN" : Bool := TRUE;
      "X14-2.ANODE NG BOX LOCK UP" : Bool := FALSE;
      "X16-1.ANODE NG BOX NG BOX DETECT SENSOR" : Bool := TRUE;
      "X16-2.SPARE" : Bool := FALSE;
   END_VAR
BEGIN
END_DATA_BLOCK

DATA_BLOCK "BK12"   // DB291
// stored: MemoryReserve 100
   VAR
      "X10-1.ANODE NG P&P 1st BACKWARD" : Bool := FALSE;
      "X11-1.SPARE" : Bool := FALSE;
      "X12-1.ANODE NG P&P 2nd BACKWARD" : Bool := FALSE;
      "X13-1.SPARE" : Bool := FALSE;
      "X14-1.ANODE NG P&P UP" : Bool := TRUE;
      "X15-1.SPARE" : Bool := FALSE;
      "X16-1.ANODE NG P&P VACUUM PRESSURE SWITCH" : Bool := FALSE;
      "X17-1.SPARE" : Bool := FALSE;
      "X10-2.ANODE NG P&P 1st FORWARD" : Bool := FALSE;
      "X11-2.SPARE" : Bool := FALSE;
      "X12-2.ANODE NG P&P 2nd FORWARD" : Bool := FALSE;
      "X13-2.SPARE" : Bool := FALSE;
      "X14-2.ANODE NG P&P DOWN" : Bool := FALSE;
      "X15-2.SPARE" : Bool := FALSE;
      "X16-2.ANODE NG P&P ELECTRODE DETECT SENSOR" : Bool := TRUE;
      "X17-2.SPARE" : Bool := FALSE;
   END_VAR
BEGIN
END_DATA_BLOCK

DATA_BLOCK "BK13"   // DB282
// stored: MemoryReserve 100
   VAR
      "X10-1.CATHODE ALIGN TABLE Y1-AXIS LIMIT SENSOR(-)" : Bool := TRUE;
      "X11-1.CATHODE ALIGN TABLE Y1-AXIS LIMIT SENSOR(+)" : Bool := TRUE;
      "X12-1.CATHODE ALIGN TABLE X-AXIS LIMIT SENSOR(-)" : Bool := TRUE;
      "X13-1.CATHODE ALIGN TABLE X-AXIS LIMIT SENSOR(+)" : Bool := TRUE;
      "X14-1.CATHODE ALIGN TABLE Y2-AXIS LIMIT SENSOR(-)" : Bool := TRUE;
      "X15-1.CATHODE ALIGN TABLE Y2-AXIS LIMIT SENSOR(+)" : Bool := TRUE;
      "X16-1.CATHODE ALIGN TABLE ELECTRODE DETECT SENSOR" : Bool := FALSE;
      "X17-1.CATHODE ALIGN TABLE PRESSURE SWITCH" : Bool := FALSE;
      "X10-2.CATHODE ALIGN TABLE Y1-AXIS HOME SENSOR" : Bool := TRUE;
      "X11-2.SPARE" : Bool := FALSE;
      "X12-2.CATHODE ALIGN TABLE X-AXIS HOME SENSOR" : Bool := FALSE;
      "X13-2.SPARE" : Bool := FALSE;
      "X14-2.CATHODE ALIGN TABLE Y2-AXIS HOME SENSOR" : Bool := FALSE;
      "X15-2.SPARE" : Bool := FALSE;
      "X16-2.SPARE" : Bool := FALSE;
      "X17-2.SPARE" : Bool := FALSE;
   END_VAR
BEGIN
END_DATA_BLOCK

DATA_BLOCK "BK14"   // DB292
// stored: MemoryReserve 100
   VAR
      "X10-1.FIX CATHODE FRONT BACKWARD" : Bool := FALSE;
      "X11-1.STACK TABLE OUT REAR Z-AXIS LIMIT SENSOR(-)" : Bool := TRUE;
      "X12-1.FIX CATHODE REAR BACKWARD" : Bool := FALSE;
      "X13-1.STACK TABLE OUT REAR Z-AXIS LIMIT SENSOR(+)" : Bool := TRUE;
      "X14-1.FIX CATHODE DETECT SENSOR" : Bool := FALSE;
      "X15-1.SPARE" : Bool := FALSE;
      "X16-1.SPARE" : Bool := FALSE;
      "X17-1.SPARE" : Bool := FALSE;
      "X10-2.FIX CATHODE FRONT FORWARD" : Bool := TRUE;
      "X11-2.STACK TABLE OUT REAR Z-AXIS HOME SENSOR" : Bool := TRUE;
      "X12-2.FIX CATHODE REAR FORWARD" : Bool := TRUE;
      "X13-2.SPARE" : Bool := FALSE;
      "X14-2.SPARE" : Bool := FALSE;
      "X15-2.SPARE" : Bool := FALSE;
      "X16-2.SPARE" : Bool := FALSE;
      "X17-2.SPARE" : Bool := FALSE;
   END_VAR
BEGIN
END_DATA_BLOCK

DATA_BLOCK "BK15"   // DB301
// stored: MemoryReserve 100
   VAR
      "X10-1.CATHODE NG BOX FULL SENSOR" : Bool := FALSE;
      "X10-2.CATHODE NG BOX NG BOX DETECT SENSOR" : Bool := TRUE;
      "X12-1.CATHODE NG BOX LIFT DOWN" : Bool := FALSE;
      "X12-2.CATHODE NG BOX LIFT UP" : Bool := TRUE;
      "X14-1.CATHODE NG BOX LOCK DOWN" : Bool := TRUE;
      "X14-2.CATHODE NG BOX LOCK UP" : Bool := FALSE;
      "X16-1.SPARE" : Bool := FALSE;
      "X16-2.SPARE" : Bool := FALSE;
   END_VAR
BEGIN
END_DATA_BLOCK

DATA_BLOCK "BK16"   // DB300
// stored: MemoryReserve 100
   VAR
      "X10-1.CATHODE NG P&P 1st BACKWARD" : Bool := TRUE;
      "X11-1.SPARE" : Bool := FALSE;
      "X12-1.CATHODE NG P&P 2nd BACKWARD" : Bool := TRUE;
      "X13-1.SPARE" : Bool := FALSE;
      "X14-1.CATHODE NG P&P DOWN" : Bool := TRUE;
      "X15-1.SPARE" : Bool := FALSE;
      "X16-1.CATHODE NG P&P VACUUM PRESSURE SWITCH" : Bool := FALSE;
      "X17-1.SPARE" : Bool := FALSE;
      "X10-2.CATHODE NG P&P 1st FORWARD" : Bool := FALSE;
      "X11-2.SPARE" : Bool := FALSE;
      "X12-2.CATHODE NG P&P 2nd FORWARD" : Bool := FALSE;
      "X13-2.SPARE" : Bool := FALSE;
      "X14-2.CATHODE NG P&P UP" : Bool := FALSE;
      "X15-2.SPARE" : Bool := FALSE;
      "X16-2.CATHODE NG P&P ELECTRODE DETECT SENSOR" : Bool := FALSE;
      "X17-2.SPARE" : Bool := FALSE;
   END_VAR
BEGIN
END_DATA_BLOCK

DATA_BLOCK "BK17"   // DB313
// stored: MemoryReserve 100
   VAR
      "X10-1.FINAL ROLLER FRONT LIMIT SENSOR(-)" : Bool := TRUE;
      "X10-2.FINAL ROLLER FRONT HOME SENSOR" : Bool := TRUE;
      "X12-1.FINAL ROLLER FRONT LIMIT SENSOR(+)" : Bool := TRUE;
      "X12-2.SPARE" : Bool := FALSE;
      "X14-1.FINAL ROLLER REAR LIMIT SENSOR(-)" : Bool := TRUE;
      "X14-2.FINAL ROLLER REAR HOME SENSOR" : Bool := TRUE;
      "X16-1.FINAL ROLLER REAR LIMIT SENSOR(+)" : Bool := TRUE;
      "X16-2.SPARE" : Bool := FALSE;
   END_VAR
BEGIN
END_DATA_BLOCK

DATA_BLOCK "BK18"   // DB312
// stored: MemoryReserve 100
   VAR
      "X10-1.ANODE MANDREL REAR Y AXIS LIMIT SENSOR(-)" : Bool := TRUE;
      "X11-1.ANODE MANDREL REAR Y AXIS LIMIT SENSOR(+)" : Bool := TRUE;
      "X12-1.ANODE MANDREL REAR Z AXIS LIMIT SENSOR(-)" : Bool := TRUE;
      "X13-1.ANODE MANDREL REAR Z AXIS LIMIT SENSOR(+)" : Bool := TRUE;
      "X14-1.ANODE MANDREL FRONT Y AXIS LIMIT SENSOR(-)" : Bool := TRUE;
      "X15-1.ANODE MANDREL FRONT Y AXIS LIMIT SENSOR(+)" : Bool := TRUE;
      "X16-1.ANODE MANDREL FRONT Z AXIS LIMIT SENSOR(-)" : Bool := TRUE;
      "X17-1.ANODE MANDREL FRONT Z AXIS LIMIT SENSOR(+)" : Bool := TRUE;
      "X10-2.ANODE MANDREL REAR Y AXIS HOME SENSOR" : Bool := TRUE;
      "X11-2.SPARE" : Bool := FALSE;
      "X12-2.ANODE MANDREL REAR Z AXIS HOME SENSOR" : Bool := TRUE;
      "X13-2.SPARE" : Bool := FALSE;
      "X14-2.ANODE MANDREL FRONT Y AXIS HOME SENSOR" : Bool := TRUE;
      "X15-2.SPARE" : Bool := FALSE;
      "X16-2.ANODE MANDREL FRONT Z AXIS HOME SENSOR" : Bool := TRUE;
      "X17-2.SPARE" : Bool := FALSE;
   END_VAR
BEGIN
END_DATA_BLOCK

DATA_BLOCK "BK19"   // DB314
// stored: MemoryReserve 100
   VAR
      "X10-1.CATHODE MANDREL REAR Y AXIS LIMIT SENSOR(-)" : Bool := TRUE;
      "X11-1.CATHODE MANDREL REAR Y AXIS LIMIT SENSOR(+)" : Bool := TRUE;
      "X12-1.CATHODE MANDREL REAR Z AXIS LIMIT SENSOR(-)" : Bool := TRUE;
      "X13-1.CATHODE MANDREL REAR Z AXIS LIMIT SENSOR(+)" : Bool := TRUE;
      "X14-1.CATHODE MANDREL FRONT Y AXIS LIMIT SENSOR(-)" : Bool := TRUE;
      "X15-1.CATHODE MANDREL FRONT Y AXIS LIMIT SENSOR(+)" : Bool := TRUE;
      "X16-1.CATHODE MANDREL FRONT Z AXIS LIMIT SENSOR(-)" : Bool := TRUE;
      "X17-1.CATHODE MANDREL FRONT Z AXIS LIMIT SENSOR(+)" : Bool := TRUE;
      "X10-2.CATHODE MANDREL REAR Y AXIS HOME SENSOR" : Bool := TRUE;
      "X11-2.SPARE" : Bool := FALSE;
      "X12-2.CATHODE MANDREL REAR Z AXIS HOME SENSOR" : Bool := TRUE;
      "X13-2.SPARE" : Bool := FALSE;
      "X14-2.CATHODE MANDREL FRONT Y AXIS HOME SENSOR" : Bool := TRUE;
      "X15-2.SPARE" : Bool := FALSE;
      "X16-2.CATHODE MANDREL FRONT Z AXIS HOME SENSOR" : Bool := TRUE;
      "X17-2.SPARE" : Bool := FALSE;
   END_VAR
BEGIN
END_DATA_BLOCK

DATA_BLOCK "BK20"   // DB311
// stored: MemoryReserve 100
   VAR
      "X10-1.STACK TABLE Z-AXIS LIMIT SENSOR(-)" : Bool := TRUE;
      "X11-1.STACK TABLE Z-AXIS LIMIT SENSOR(+)" : Bool := TRUE;
      "X12-1.STACK TABLE GAP PAD DOWN" : Bool := TRUE;
      "X13-1.STACK TABLE GAP PAD UP" : Bool := FALSE;
      "X14-1.STACK TABLE OUT FRONT Z-AXIS LIMIT SENSOR(-)" : Bool := TRUE;
      "X15-1.STACK TABLE OUT FRONT Z-AXIS LIMIT SENSOR(+)" : Bool := TRUE;
      "X16-1.STACK TABLE VACUUM PRESSURE SWITCH" : Bool := FALSE;
      "X17-1.SPARE" : Bool := FALSE;
      "X10-2.STACK TABLE Z-AXIS HOME SENSOR" : Bool := TRUE;
      "X11-2.SPARE" : Bool := FALSE;
      "X12-2.SPARE" : Bool := FALSE;
      "X13-2.SPARE" : Bool := FALSE;
      "X14-2.STACK TABLE OUT FRONT Z-AXIS HOME SENSOR" : Bool := TRUE;
      "X15-2.SPARE" : Bool := FALSE;
      "X16-2.STACK TABLE ELECTRODE DETECT SENSOR" : Bool := FALSE;
      "X17-2.SPARE" : Bool := FALSE;
   END_VAR
BEGIN
END_DATA_BLOCK

DATA_BLOCK "BK21"   // DB249
// stored: MemoryReserve 100
   VAR
      "X10-1.SEPA CLAMP&CUTTER X-AXIS LIMIT SENSOR(-)" : Bool := TRUE;
      "X10-2.SEPA CLAMP&CUTTER X-AXIS HOME SENSOR" : Bool := TRUE;
      "X12-1.SEPA CLAMP&CUTTER X-AXIS LIMIT SENSOR(+)" : Bool := TRUE;
      "X12-2.SPARE" : Bool := FALSE;
      "X14-1.SEPA GRIPPER X-AXIS LIMIT SENSOR(-)" : Bool := TRUE;
      "X14-2.SEPA GRIPPER X-AXIS HOME SENSOR" : Bool := TRUE;
      "X16-1.SEPA GRIPPER X-AXIS LIMIT SENSOR(+)" : Bool := TRUE;
      "X16-2.SPARE" : Bool := FALSE;
   END_VAR
BEGIN
END_DATA_BLOCK

DATA_BLOCK "BK22"   // DB274
// stored: MemoryReserve 100
   VAR
      "X10-1.SEPA GRIPPER CLAMP OPEN" : Bool := TRUE;
      "X11-1.SPARE" : Bool := FALSE;
      "X12-1.SEPA GRIPPER CLAMP DETECT SENSOR" : Bool := TRUE;
      "X13-1.SEPA GRIPPER BACKWARD" : Bool := FALSE;
      "X14-1.SEPA GRIPPER C-AXIS LIMIT SENSOR(-)" : Bool := FALSE;
      "X15-1.SEPA GRIPPER C-AXIS LIMIT SENSOR(+)" : Bool := TRUE;
      "X16-1.SEPA GRIPPER Z-AXIS LIMIT SENSOR(-)" : Bool := TRUE;
      "X17-1.SEPA GRIPPER Z-AXIS LIMIT SENSOR(+)" : Bool := TRUE;
      "X10-2.SEPA GRIPPER CLAMP CLOSE" : Bool := FALSE;
      "X11-2.SPARE" : Bool := FALSE;
      "X12-2.SPARE" : Bool := FALSE;
      "X13-2.SEPA GRIPPER FORWARD" : Bool := FALSE;
      "X14-2.SEPA GRIPPER C-AXIS HOME SENSOR" : Bool := FALSE;
      "X15-2.SPARE" : Bool := FALSE;
      "X16-2.SEPA GRIPPER Z-AXIS HOME SENSOR" : Bool := TRUE;
      "X17-2.SPARE" : Bool := FALSE;
   END_VAR
BEGIN
END_DATA_BLOCK

DATA_BLOCK "BK23"   // DB142
// stored: MemoryReserve 100
   VAR
      "X10-1.SEPA CLAMP&CUTTER Z-AXIS LIMIT SENSOR(-)" : Bool := TRUE;
      "X11-1.SEPA CLAMP&CUTTER Z-AXIS LIMIT SENSOR(+)" : Bool := TRUE;
      "X12-1.SEPA CUTTER UP" : Bool := FALSE;
      "X13-1.SPARE" : Bool := FALSE;
      "X14-1.SPARE" : Bool := FALSE;
      "X15-1.SPARE" : Bool := FALSE;
      "X16-1.SEPA DETECT SENSOR" : Bool := FALSE;
      "X17-1.SPARE" : Bool := FALSE;
      "X10-2.CLAMP&CUTTER Z-AXIS HOME SENSOR" : Bool := TRUE;
      "X11-2.SPARE" : Bool := FALSE;
      "X12-2.SEPA CUTTER DOWN" : Bool := TRUE;
      "X13-2.SPARE" : Bool := FALSE;
      "X14-2.SPARE" : Bool := FALSE;
      "X15-2.SPARE" : Bool := FALSE;
      "X16-2.SPARE" : Bool := FALSE;
      "X17-2.SPARE" : Bool := FALSE;
   END_VAR
BEGIN
END_DATA_BLOCK

DATA_BLOCK "BK24"   // DB238
// stored: MemoryReserve 100
   VAR
      "X10-1.SEPA CLAMP TOP REAR UP" : Bool := FALSE;
      "X11-1.SPARE" : Bool := FALSE;
      "X12-1.SEPA CLAMP TOP FRONT UP" : Bool := FALSE;
      "X13-1.SPARE" : Bool := FALSE;
      "X14-1.SEPA CLAMP BTM REAR UP" : Bool := TRUE;
      "X15-1.SPARE" : Bool := FALSE;
      "X16-1.SEPA CLAMP BTM FRONT UP" : Bool := TRUE;
      "X17-1.SPARE" : Bool := FALSE;
      "X10-2.SEPA CLAMP TOP REAR DOWN" : Bool := TRUE;
      "X11-2.SPARE" : Bool := FALSE;
      "X12-2.SEPA CLAMP TOP FRONT DOWN" : Bool := TRUE;
      "X13-2.SPARE" : Bool := FALSE;
      "X14-2.SEPA CLAMP BTM REAR DOWN" : Bool := FALSE;
      "X15-2.SPARE" : Bool := FALSE;
      "X16-2.SEPA CLAMP BTM FRONT DOWN" : Bool := FALSE;
      "X17-2.SPARE" : Bool := FALSE;
   END_VAR
BEGIN
END_DATA_BLOCK

DATA_BLOCK "BK25"   // DB273
// stored: MemoryReserve 100
   VAR
      "X10-1.JR WINDER REAR Y-AXIS LIMIT SENSOR(-)" : Bool := TRUE;
      "X10-2.JR WINDER REAR Y-AXIS HOME SENSOR" : Bool := FALSE;
      "X12-1.JR WINDER REAR Y-AXIS LIMIT SENSOR(+)" : Bool := TRUE;
      "X12-2.SPARE" : Bool := FALSE;
      "X14-1.JR WINDER FRONT Y-AXIS LIMIT SENSOR(-)" : Bool := TRUE;
      "X14-2.JR WINDER FRONT Y-AXIS HOME SENSOR" : Bool := TRUE;
      "X16-1.JR WINDER FRONT Y-AXIS LIMIT SENSOR(+)" : Bool := TRUE;
      "X16-2.SPARE" : Bool := FALSE;
   END_VAR
BEGIN
END_DATA_BLOCK

DATA_BLOCK "BK26"   // DB260
// stored: MemoryReserve 100
   VAR
      "X10-1.JR WINDER B-AXIS HOME SENSOR" : Bool := TRUE;
      "X11-1.JR WINDER CLAMP TOP REAR UP/DOWN" : Bool := FALSE;
      "X12-1.MAIN VALVE DIGITAL PRESSURE SWITCH OUT1" : Bool := FALSE;
      "X13-1.JR WINDER CLAMP TOP FRONT UP/DOWN" : Bool := FALSE;
      "X14-1.SPARE" : Bool := FALSE;
      "X15-1.JR WINDER CLAMP TOP REAR PRESSURE SWITCH" : Bool := FALSE;
      "X16-1.SPARE" : Bool := FALSE;
      "X17-1.SPARE" : Bool := FALSE;
      "X10-2.SPARE" : Bool := FALSE;
      "X11-2.SPARE" : Bool := FALSE;
      "X12-2.MAIN VALVE DIGITAL PRESSURE SWITCH OUT2" : Bool := FALSE;
      "X13-2.SPARE" : Bool := FALSE;
      "X14-2.SPARE" : Bool := FALSE;
      "X15-2.JR WINDER CLAMP TOP FRONT PRESSURE SWITCH" : Bool := FALSE;
      "X16-2.SPARE" : Bool := FALSE;
      "X17-2.SPARE" : Bool := FALSE;
   END_VAR
BEGIN
END_DATA_BLOCK

DATA_BLOCK "BK27"   // DB255
// stored: MemoryReserve 100
   VAR
      "X10-1.SPARE" : Bool := FALSE;
      "X11-1.JR WINDER CLAMP BTM REAR UP/DOWN" : Bool := FALSE;
      "X12-1.SPARE" : Bool := FALSE;
      "X13-1.JR WINDER CLAMP BTM FRONT UP/DOWN" : Bool := FALSE;
      "X14-1.SPARE" : Bool := FALSE;
      "X15-1.JR WINDER CLAMP FRONT TOP PRESSURE SWITCH" : Bool := FALSE;
      "X16-1.JR WINDER STACK DETECT SENSOR" : Bool := FALSE;
      "X17-1.SPARE" : Bool := FALSE;
      "X10-2.SPARE" : Bool := FALSE;
      "X11-2.SPARE" : Bool := FALSE;
      "X12-2.SPARE" : Bool := FALSE;
      "X13-2.SPARE" : Bool := FALSE;
      "X14-2.SPARE" : Bool := FALSE;
      "X15-2.JR WINDER CLAMP FRONT BTM PRESSURE SWITCH" : Bool := FALSE;
      "X16-2.SPARE" : Bool := FALSE;
      "X17-2.SPARE" : Bool := FALSE;
   END_VAR
BEGIN
END_DATA_BLOCK

DATA_BLOCK "BK28"   // DB272
// stored: MemoryReserve 100
   VAR
      "X10-1.PUSHER ROLLER Z-AXIS LIMIT SENSOR(-)" : Bool := FALSE;
      "X10-2.PUSHER ROLLER Z-AXIS HOME SENSOR" : Bool := FALSE;
      "X12-1.PUSH ROLLER BACKWARD" : Bool := FALSE;
      "X12-2.PUSH ROLLER FORWARD" : Bool := FALSE;
      "X14-1.SPARE" : Bool := FALSE;
      "X14-2.SPARE" : Bool := FALSE;
      "X16-1.PUSHER ROLLER Z-AXIS LIMIT SENSOR(+)" : Bool := FALSE;
      "X16-2.SPARE" : Bool := FALSE;
   END_VAR
BEGIN
END_DATA_BLOCK

DATA_BLOCK "BK29"   // DB280
// stored: MemoryReserve 100
   VAR
      "X10-1.SUCTION PAD TOP LEFT VACUUM ON" : Bool := FALSE;
      "X10-2.SUCTION PAD TOP LEFT VACUUM OFF" : Bool := FALSE;
      "X12-1.SUCTION PAD TOP RIGHT VACUUM ON" : Bool := FALSE;
      "X12-2.SUCTION PAD TOP RIGHT VACUUM OFF" : Bool := FALSE;
      "X14-1.SUCTION PAD BTM LEFT VACUUM ON" : Bool := FALSE;
      "X14-2.SUCTION PAD BTM LEFT VACUUM OFF" : Bool := FALSE;
      "X16-1.SUCTION PAD BTM RIGHT VACUUM ON" : Bool := FALSE;
      "X16-2.SUCTION PAD BTM RIGHT VACUUM OFF" : Bool := FALSE;
   END_VAR
BEGIN
END_DATA_BLOCK

DATA_BLOCK "BK30"   // DB237
// stored: MemoryReserve 100
   VAR
      "X10-1.SUCTION PAD TOP TAPE VACUUM ON" : Bool := FALSE;
      "X10-2.SUCTION PAD TOP TAPE VACUUM OFF" : Bool := FALSE;
      "X12-1.SUCTION PAD BTM TAPE VACUUM ON" : Bool := FALSE;
      "X12-2.SUCTION PAD BTM TAPE VACUUM OFF" : Bool := FALSE;
      "X14-1.STACK TABLE VACUUM ON" : Bool := FALSE;
      "X14-2.STACK TABLE VACUUM OFF" : Bool := FALSE;
      "X16-1.SPARE" : Bool := FALSE;
      "X16-2.SPARE" : Bool := FALSE;
   END_VAR
BEGIN
END_DATA_BLOCK

DATA_BLOCK "BK31"   // DB279
// stored: MemoryReserve 100
   VAR
      "X10-1.ANODE MAIN P&P1-1 VACUUM ON" : Bool := FALSE;
      "X10-2.ANODE MAIN P&P1-1 VACUUM OFF" : Bool := FALSE;
      "X12-1.ANODE MAIN P&P2-1 VACUUM ON" : Bool := FALSE;
      "X12-2.ANODE MAIN P&P2-1 VACUUM OFF" : Bool := FALSE;
      "X14-1.ANODE MAIN NG P&P VACUUM ON" : Bool := FALSE;
      "X14-2.ANODE MAIN NG P&P VACUUM OFF" : Bool := FALSE;
      "X16-1.ANODE ALIGN TABLE VACUUM ON" : Bool := FALSE;
      "X16-2.ANODE ALIGN TABLE VACUUM OFF" : Bool := FALSE;
   END_VAR
BEGIN
END_DATA_BLOCK

DATA_BLOCK "BK32"   // DB259
// stored: MemoryReserve 100
   VAR
      "X10-1.CATHODE MAIN P&P1-1 VACUUM ON" : Bool := FALSE;
      "X10-2.CATHODE MAIN P&P1-1 VACUUM OFF" : Bool := FALSE;
      "X12-1.CATHODE MAIN P&P2-1 VACUUM ON" : Bool := FALSE;
      "X12-2.CATHODE MAIN P&P2-1 VACUUM OFF" : Bool := FALSE;
      "X14-1.CATHODE MAIN NG P&P VACUUM ON" : Bool := FALSE;
      "X14-2.CATHODE MAIN NG P&P VACUUM OFF" : Bool := FALSE;
      "X16-1.CATHODE ALIGN TABLE VACUUM ON" : Bool := FALSE;
      "X16-2.CATHODE ALIGN TABLE VACUUM OFF" : Bool := FALSE;
   END_VAR
BEGIN
END_DATA_BLOCK

DATA_BLOCK "BK33"   // DB236
// stored: MemoryReserve 100
   VAR
      "X10-1.ANODE MAIN P&P1-2 VACUUM ON" : Bool := FALSE;
      "X10-2.ANODE MAIN P&P1-2 VACUUM OFF" : Bool := FALSE;
      "X12-1.CATHODE MAIN P&P1-2 VACUUM ON" : Bool := FALSE;
      "X12-2.CATHODE MAIN P&P1-2 VACUUM OFF" : Bool := FALSE;
      "X14-1.ANODE MAIN P&P2-2 VACUUM ON" : Bool := FALSE;
      "X14-2.ANODE MAIN P&P2-2 VACUUM OFF" : Bool := FALSE;
      "X16-1.CATHODE MAIN P&P2-2 VACUUM ON" : Bool := FALSE;
      "X16-2.CATHODE MAIN P&P2-2 VACUUM OFF" : Bool := FALSE;
   END_VAR
BEGIN
END_DATA_BLOCK

DATA_BLOCK "BK34"   // DB309
// stored: MemoryReserve 100
   VAR
      "X10-1.UNWINDER #1 RADIUS MEASURE" : Bool := FALSE;
      "X11-1.UNWINDER #2 RADIUS MEASURE" : Bool := FALSE;
      "X12-1.SPARE" : Bool := FALSE;
      "X12-2.SPARE" : Bool := FALSE;
      "X14-1.SPARE" : Bool := FALSE;
      "X14-2.SPARE" : Bool := FALSE;
      "X16-1.SPARE" : Bool := FALSE;
      "X16-2.SPARE" : Bool := FALSE;
   END_VAR
BEGIN
END_DATA_BLOCK

DATA_BLOCK "MotorStarterHMI"   // DB212
// stored: MemoryReserve 100
   VAR
      unitMotorstarter : Array[0.."NO_OF_UNITS"] of "typeEmMotorStarterInterface";
   END_VAR
BEGIN
   unitMotorstarter[0].EMmotorstarter[0].et200SpMotorstarterCurrent[0..1] := 0.0;
   unitMotorstarter[0].EMmotorstarter[1].et200SpMotorstarterCurrent[0..1] := 0.0;
   unitMotorstarter[0].EMmotorstarter[2].et200SpMotorstarterCurrent[0..1] := 0.0;
   unitMotorstarter[0].EMmotorstarter[3].et200SpMotorstarterCurrent[0..1] := 0.0;
   unitMotorstarter[0].EMmotorstarter[4].et200SpMotorstarterCurrent[0..1] := 0.0;
   unitMotorstarter[0].EMmotorstarter[5].et200SpMotorstarterCurrent[0..1] := 0.0;
   unitMotorstarter[0].EMmotorstarter[6].et200SpMotorstarterCurrent[0..1] := 0.0;
   unitMotorstarter[0].EMmotorstarter[7].et200SpMotorstarterCurrent[0..1] := 0.0;
   unitMotorstarter[0].EMmotorstarter[0].et200SpMotorstarterInputs[0..1].readyAutomatic := FALSE;
   unitMotorstarter[0].EMmotorstarter[1].et200SpMotorstarterInputs[0..1].readyAutomatic := FALSE;
   unitMotorstarter[0].EMmotorstarter[2].et200SpMotorstarterInputs[0..1].readyAutomatic := FALSE;
   unitMotorstarter[0].EMmotorstarter[3].et200SpMotorstarterInputs[0..1].readyAutomatic := FALSE;
   unitMotorstarter[0].EMmotorstarter[4].et200SpMotorstarterInputs[0..1].readyAutomatic := FALSE;
   unitMotorstarter[0].EMmotorstarter[5].et200SpMotorstarterInputs[0..1].readyAutomatic := FALSE;
   unitMotorstarter[0].EMmotorstarter[6].et200SpMotorstarterInputs[0..1].readyAutomatic := FALSE;
   unitMotorstarter[0].EMmotorstarter[7].et200SpMotorstarterInputs[0..1].readyAutomatic := FALSE;
   unitMotorstarter[0].EMmotorstarter[0].et200SpMotorstarterInputs[0..1].motorOn := FALSE;
   unitMotorstarter[0].EMmotorstarter[1].et200SpMotorstarterInputs[0..1].motorOn := FALSE;
   unitMotorstarter[0].EMmotorstarter[2].et200SpMotorstarterInputs[0..1].motorOn := FALSE;
   unitMotorstarter[0].EMmotorstarter[3].et200SpMotorstarterInputs[0..1].motorOn := FALSE;
   unitMotorstarter[0].EMmotorstarter[4].et200SpMotorstarterInputs[0..1].motorOn := FALSE;
   unitMotorstarter[0].EMmotorstarter[5].et200SpMotorstarterInputs[0..1].motorOn := FALSE;
   unitMotorstarter[0].EMmotorstarter[6].et200SpMotorstarterInputs[0..1].motorOn := FALSE;
   unitMotorstarter[0].EMmotorstarter[7].et200SpMotorstarterInputs[0..1].motorOn := FALSE;
   unitMotorstarter[0].EMmotorstarter[0].et200SpMotorstarterInputs[0..1].groupFault := FALSE;
   unitMotorstarter[0].EMmotorstarter[1].et200SpMotorstarterInputs[0..1].groupFault := FALSE;
   unitMotorstarter[0].EMmotorstarter[2].et200SpMotorstarterInputs[0..1].groupFault := FALSE;
   unitMotorstarter[0].EMmotorstarter[3].et200SpMotorstarterInputs[0..1].groupFault := FALSE;
   unitMotorstarter[0].EMmotorstarter[4].et200SpMotorstarterInputs[0..1].groupFault := FALSE;
   unitMotorstarter[0].EMmotorstarter[5].et200SpMotorstarterInputs[0..1].groupFault := FALSE;
   unitMotorstarter[0].EMmotorstarter[6].et200SpMotorstarterInputs[0..1].groupFault := FALSE;
   unitMotorstarter[0].EMmotorstarter[7].et200SpMotorstarterInputs[0..1].groupFault := FALSE;
   unitMotorstarter[0].EMmotorstarter[0].et200SpMotorstarterInputs[0..1].groupWarning := FALSE;
   unitMotorstarter[0].EMmotorstarter[1].et200SpMotorstarterInputs[0..1].groupWarning := FALSE;
   unitMotorstarter[0].EMmotorstarter[2].et200SpMotorstarterInputs[0..1].groupWarning := FALSE;
   unitMotorstarter[0].EMmotorstarter[3].et200SpMotorstarterInputs[0..1].groupWarning := FALSE;
   unitMotorstarter[0].EMmotorstarter[4].et200SpMotorstarterInputs[0..1].groupWarning := FALSE;
   unitMotorstarter[0].EMmotorstarter[5].et200SpMotorstarterInputs[0..1].groupWarning := FALSE;
   unitMotorstarter[0].EMmotorstarter[6].et200SpMotorstarterInputs[0..1].groupWarning := FALSE;
   unitMotorstarter[0].EMmotorstarter[7].et200SpMotorstarterInputs[0..1].groupWarning := FALSE;
   unitMotorstarter[0].EMmotorstarter[0].et200SpMotorstarterInputs[0..1].input1 := FALSE;
   unitMotorstarter[0].EMmotorstarter[1].et200SpMotorstarterInputs[0..1].input1 := FALSE;
   unitMotorstarter[0].EMmotorstarter[2].et200SpMotorstarterInputs[0..1].input1 := FALSE;
   unitMotorstarter[0].EMmotorstarter[3].et200SpMotorstarterInputs[0..1].input1 := FALSE;
   unitMotorstarter[0].EMmotorstarter[4].et200SpMotorstarterInputs[0..1].input1 := FALSE;
   unitMotorstarter[0].EMmotorstarter[5].et200SpMotorstarterInputs[0..1].input1 := FALSE;
   unitMotorstarter[0].EMmotorstarter[6].et200SpMotorstarterInputs[0..1].input1 := FALSE;
   unitMotorstarter[0].EMmotorstarter[7].et200SpMotorstarterInputs[0..1].input1 := FALSE;
   unitMotorstarter[0].EMmotorstarter[0].et200SpMotorstarterInputs[0..1].input2 := FALSE;
   unitMotorstarter[0].EMmotorstarter[1].et200SpMotorstarterInputs[0..1].input2 := FALSE;
   unitMotorstarter[0].EMmotorstarter[2].et200SpMotorstarterInputs[0..1].input2 := FALSE;
   unitMotorstarter[0].EMmotorstarter[3].et200SpMotorstarterInputs[0..1].input2 := FALSE;
   unitMotorstarter[0].EMmotorstarter[4].et200SpMotorstarterInputs[0..1].input2 := FALSE;
   unitMotorstarter[0].EMmotorstarter[5].et200SpMotorstarterInputs[0..1].input2 := FALSE;
   unitMotorstarter[0].EMmotorstarter[6].et200SpMotorstarterInputs[0..1].input2 := FALSE;
   unitMotorstarter[0].EMmotorstarter[7].et200SpMotorstarterInputs[0..1].input2 := FALSE;
   unitMotorstarter[0].EMmotorstarter[0].et200SpMotorstarterInputs[0..1].input3 := FALSE;
   unitMotorstarter[0].EMmotorstarter[1].et200SpMotorstarterInputs[0..1].input3 := FALSE;
   unitMotorstarter[0].EMmotorstarter[2].et200SpMotorstarterInputs[0..1].input3 := FALSE;
   unitMotorstarter[0].EMmotorstarter[3].et200SpMotorstarterInputs[0..1].input3 := FALSE;
   unitMotorstarter[0].EMmotorstarter[4].et200SpMotorstarterInputs[0..1].input3 := FALSE;
   unitMotorstarter[0].EMmotorstarter[5].et200SpMotorstarterInputs[0..1].input3 := FALSE;
   unitMotorstarter[0].EMmotorstarter[6].et200SpMotorstarterInputs[0..1].input3 := FALSE;
   unitMotorstarter[0].EMmotorstarter[7].et200SpMotorstarterInputs[0..1].input3 := FALSE;
   unitMotorstarter[0].EMmotorstarter[0].et200SpMotorstarterInputs[0..1].inputLocalCtrl := FALSE;
   unitMotorstarter[0].EMmotorstarter[1].et200SpMotorstarterInputs[0..1].inputLocalCtrl := FALSE;
   unitMotorstarter[0].EMmotorstarter[2].et200SpMotorstarterInputs[0..1].inputLocalCtrl := FALSE;
   unitMotorstarter[0].EMmotorstarter[3].et200SpMotorstarterInputs[0..1].inputLocalCtrl := FALSE;
   unitMotorstarter[0].EMmotorstarter[4].et200SpMotorstarterInputs[0..1].inputLocalCtrl := FALSE;
   unitMotorstarter[0].EMmotorstarter[5].et200SpMotorstarterInputs[0..1].inputLocalCtrl := FALSE;
   unitMotorstarter[0].EMmotorstarter[6].et200SpMotorstarterInputs[0..1].inputLocalCtrl := FALSE;
   unitMotorstarter[0].EMmotorstarter[7].et200SpMotorstarterInputs[0..1].inputLocalCtrl := FALSE;
   unitMotorstarter[0].EMmotorstarter[0].et200SpMotorstarterInputs[0..1].iActBit0 := FALSE;
   unitMotorstarter[0].EMmotorstarter[1].et200SpMotorstarterInputs[0..1].iActBit0 := FALSE;
   unitMotorstarter[0].EMmotorstarter[2].et200SpMotorstarterInputs[0..1].iActBit0 := FALSE;
   unitMotorstarter[0].EMmotorstarter[3].et200SpMotorstarterInputs[0..1].iActBit0 := FALSE;
   unitMotorstarter[0].EMmotorstarter[4].et200SpMotorstarterInputs[0..1].iActBit0 := FALSE;
   unitMotorstarter[0].EMmotorstarter[5].et200SpMotorstarterInputs[0..1].iActBit0 := FALSE;
   unitMotorstarter[0].EMmotorstarter[6].et200SpMotorstarterInputs[0..1].iActBit0 := FALSE;
   unitMotorstarter[0].EMmotorstarter[7].et200SpMotorstarterInputs[0..1].iActBit0 := FALSE;
   unitMotorstarter[0].EMmotorstarter[0].et200SpMotorstarterInputs[0..1].iActBit1 := FALSE;
   unitMotorstarter[0].EMmotorstarter[1].et200SpMotorstarterInputs[0..1].iActBit1 := FALSE;
   unitMotorstarter[0].EMmotorstarter[2].et200SpMotorstarterInputs[0..1].iActBit1 := FALSE;
   unitMotorstarter[0].EMmotorstarter[3].et200SpMotorstarterInputs[0..1].iActBit1 := FALSE;
   unitMotorstarter[0].EMmotorstarter[4].et200SpMotorstarterInputs[0..1].iActBit1 := FALSE;
   unitMotorstarter[0].EMmotorstarter[5].et200SpMotorstarterInputs[0..1].iActBit1 := FALSE;
   unitMotorstarter[0].EMmotorstarter[6].et200SpMotorstarterInputs[0..1].iActBit1 := FALSE;
   unitMotorstarter[0].EMmotorstarter[7].et200SpMotorstarterInputs[0..1].iActBit1 := FALSE;
   unitMotorstarter[0].EMmotorstarter[0].et200SpMotorstarterInputs[0..1].iActBit2 := FALSE;
   unitMotorstarter[0].EMmotorstarter[1].et200SpMotorstarterInputs[0..1].iActBit2 := FALSE;
   unitMotorstarter[0].EMmotorstarter[2].et200SpMotorstarterInputs[0..1].iActBit2 := FALSE;
   unitMotorstarter[0].EMmotorstarter[3].et200SpMotorstarterInputs[0..1].iActBit2 := FALSE;
   unitMotorstarter[0].EMmotorstarter[4].et200SpMotorstarterInputs[0..1].iActBit2 := FALSE;
   unitMotorstarter[0].EMmotorstarter[5].et200SpMotorstarterInputs[0..1].iActBit2 := FALSE;
   unitMotorstarter[0].EMmotorstarter[6].et200SpMotorstarterInputs[0..1].iActBit2 := FALSE;
   unitMotorstarter[0].EMmotorstarter[7].et200SpMotorstarterInputs[0..1].iActBit2 := FALSE;
   unitMotorstarter[0].EMmotorstarter[0].et200SpMotorstarterInputs[0..1].iActBit3 := FALSE;
   unitMotorstarter[0].EMmotorstarter[1].et200SpMotorstarterInputs[0..1].iActBit3 := FALSE;
   unitMotorstarter[0].EMmotorstarter[2].et200SpMotorstarterInputs[0..1].iActBit3 := FALSE;
   unitMotorstarter[0].EMmotorstarter[3].et200SpMotorstarterInputs[0..1].iActBit3 := FALSE;
   unitMotorstarter[0].EMmotorstarter[4].et200SpMotorstarterInputs[0..1].iActBit3 := FALSE;
   unitMotorstarter[0].EMmotorstarter[5].et200SpMotorstarterInputs[0..1].iActBit3 := FALSE;
   unitMotorstarter[0].EMmotorstarter[6].et200SpMotorstarterInputs[0..1].iActBit3 := FALSE;
   unitMotorstarter[0].EMmotorstarter[7].et200SpMotorstarterInputs[0..1].iActBit3 := FALSE;
   unitMotorstarter[0].EMmotorstarter[0].et200SpMotorstarterInputs[0..1].iActBit4 := FALSE;
   unitMotorstarter[0].EMmotorstarter[1].et200SpMotorstarterInputs[0..1].iActBit4 := FALSE;
   unitMotorstarter[0].EMmotorstarter[2].et200SpMotorstarterInputs[0..1].iActBit4 := FALSE;
   unitMotorstarter[0].EMmotorstarter[3].et200SpMotorstarterInputs[0..1].iActBit4 := FALSE;
   unitMotorstarter[0].EMmotorstarter[4].et200SpMotorstarterInputs[0..1].iActBit4 := FALSE;
   unitMotorstarter[0].EMmotorstarter[5].et200SpMotorstarterInputs[0..1].iActBit4 := FALSE;
   unitMotorstarter[0].EMmotorstarter[6].et200SpMotorstarterInputs[0..1].iActBit4 := FALSE;
   unitMotorstarter[0].EMmotorstarter[7].et200SpMotorstarterInputs[0..1].iActBit4 := FALSE;
   unitMotorstarter[0].EMmotorstarter[0].et200SpMotorstarterInputs[0..1].iActBit5 := FALSE;
   unitMotorstarter[0].EMmotorstarter[1].et200SpMotorstarterInputs[0..1].iActBit5 := FALSE;
   unitMotorstarter[0].EMmotorstarter[2].et200SpMotorstarterInputs[0..1].iActBit5 := FALSE;
   unitMotorstarter[0].EMmotorstarter[3].et200SpMotorstarterInputs[0..1].iActBit5 := FALSE;
   unitMotorstarter[0].EMmotorstarter[4].et200SpMotorstarterInputs[0..1].iActBit5 := FALSE;
   unitMotorstarter[0].EMmotorstarter[5].et200SpMotorstarterInputs[0..1].iActBit5 := FALSE;
   unitMotorstarter[0].EMmotorstarter[6].et200SpMotorstarterInputs[0..1].iActBit5 := FALSE;
   unitMotorstarter[0].EMmotorstarter[7].et200SpMotorstarterInputs[0..1].iActBit5 := FALSE;
   unitMotorstarter[0].EMmotorstarter[0].et200SpMotorstarterInputs[0..1].manualOperating := FALSE;
   unitMotorstarter[0].EMmotorstarter[1].et200SpMotorstarterInputs[0..1].manualOperating := FALSE;
   unitMotorstarter[0].EMmotorstarter[2].et200SpMotorstarterInputs[0..1].manualOperating := FALSE;
   unitMotorstarter[0].EMmotorstarter[3].et200SpMotorstarterInputs[0..1].manualOperating := FALSE;
   unitMotorstarter[0].EMmotorstarter[4].et200SpMotorstarterInputs[0..1].manualOperating := FALSE;
   unitMotorstarter[0].EMmotorstarter[5].et200SpMotorstarterInputs[0..1].manualOperating := FALSE;
   unitMotorstarter[0].EMmotorstarter[6].et200SpMotorstarterInputs[0..1].manualOperating := FALSE;
   unitMotorstarter[0].EMmotorstarter[7].et200SpMotorstarterInputs[0..1].manualOperating := FALSE;
   unitMotorstarter[0].EMmotorstarter[0].et200SpMotorstarterInputs[0..1].spare1 := FALSE;
   unitMotorstarter[0].EMmotorstarter[1].et200SpMotorstarterInputs[0..1].spare1 := FALSE;
   unitMotorstarter[0].EMmotorstarter[2].et200SpMotorstarterInputs[0..1].spare1 := FALSE;
   unitMotorstarter[0].EMmotorstarter[3].et200SpMotorstarterInputs[0..1].spare1 := FALSE;
   unitMotorstarter[0].EMmotorstarter[4].et200SpMotorstarterInputs[0..1].spare1 := FALSE;
   unitMotorstarter[0].EMmotorstarter[5].et200SpMotorstarterInputs[0..1].spare1 := FALSE;
   unitMotorstarter[0].EMmotorstarter[6].et200SpMotorstarterInputs[0..1].spare1 := FALSE;
   unitMotorstarter[0].EMmotorstarter[7].et200SpMotorstarterInputs[0..1].spare1 := FALSE;
   unitMotorstarter[0].EMmotorstarter[0].et200SpMotorstarterInputs[0..1].readyStartOn := FALSE;
   unitMotorstarter[0].EMmotorstarter[1].et200SpMotorstarterInputs[0..1].readyStartOn := FALSE;
   unitMotorstarter[0].EMmotorstarter[2].et200SpMotorstarterInputs[0..1].readyStartOn := FALSE;
   unitMotorstarter[0].EMmotorstarter[3].et200SpMotorstarterInputs[0..1].readyStartOn := FALSE;
   unitMotorstarter[0].EMmotorstarter[4].et200SpMotorstarterInputs[0..1].readyStartOn := FALSE;
   unitMotorstarter[0].EMmotorstarter[5].et200SpMotorstarterInputs[0..1].readyStartOn := FALSE;
   unitMotorstarter[0].EMmotorstarter[6].et200SpMotorstarterInputs[0..1].readyStartOn := FALSE;
   unitMotorstarter[0].EMmotorstarter[7].et200SpMotorstarterInputs[0..1].readyStartOn := FALSE;
   unitMotorstarter[0].EMmotorstarter[0].et200SpMotorstarterInputs[0..1].motorOnRight := FALSE;
   unitMotorstarter[0].EMmotorstarter[1].et200SpMotorstarterInputs[0..1].motorOnRight := FALSE;
   unitMotorstarter[0].EMmotorstarter[2].et200SpMotorstarterInputs[0..1].motorOnRight := FALSE;
   unitMotorstarter[0].EMmotorstarter[3].et200SpMotorstarterInputs[0..1].motorOnRight := FALSE;
   unitMotorstarter[0].EMmotorstarter[4].et200SpMotorstarterInputs[0..1].motorOnRight := FALSE;
   unitMotorstarter[0].EMmotorstarter[5].et200SpMotorstarterInputs[0..1].motorOnRight := FALSE;
   unitMotorstarter[0].EMmotorstarter[6].et200SpMotorstarterInputs[0..1].motorOnRight := FALSE;
   unitMotorstarter[0].EMmotorstarter[7].et200SpMotorstarterInputs[0..1].motorOnRight := FALSE;
   unitMotorstarter[0].EMmotorstarter[0].et200SpMotorstarterInputs[0..1].motorOnLeft := FALSE;
   unitMotorstarter[0].EMmotorstarter[1].et200SpMotorstarterInputs[0..1].motorOnLeft := FALSE;
   unitMotorstarter[0].EMmotorstarter[2].et200SpMotorstarterInputs[0..1].motorOnLeft := FALSE;
   unitMotorstarter[0].EMmotorstarter[3].et200SpMotorstarterInputs[0..1].motorOnLeft := FALSE;
   unitMotorstarter[0].EMmotorstarter[4].et200SpMotorstarterInputs[0..1].motorOnLeft := FALSE;
   unitMotorstarter[0].EMmotorstarter[5].et200SpMotorstarterInputs[0..1].motorOnLeft := FALSE;
   unitMotorstarter[0].EMmotorstarter[6].et200SpMotorstarterInputs[0..1].motorOnLeft := FALSE;
   unitMotorstarter[0].EMmotorstarter[7].et200SpMotorstarterInputs[0..1].motorOnLeft := FALSE;
   unitMotorstarter[0].EMmotorstarter[0].et200SpMotorstarterInputs[0..1].quickstopActive := FALSE;
   unitMotorstarter[0].EMmotorstarter[1].et200SpMotorstarterInputs[0..1].quickstopActive := FALSE;
   unitMotorstarter[0].EMmotorstarter[2].et200SpMotorstarterInputs[0..1].quickstopActive := FALSE;
   unitMotorstarter[0].EMmotorstarter[3].et200SpMotorstarterInputs[0..1].quickstopActive := FALSE;
   unitMotorstarter[0].EMmotorstarter[4].et200SpMotorstarterInputs[0..1].quickstopActive := FALSE;
   unitMotorstarter[0].EMmotorstarter[5].et200SpMotorstarterInputs[0..1].quickstopActive := FALSE;
   unitMotorstarter[0].EMmotorstarter[6].et200SpMotorstarterInputs[0..1].quickstopActive := FALSE;
   unitMotorstarter[0].EMmotorstarter[7].et200SpMotorstarterInputs[0..1].quickstopActive := FALSE;
   unitMotorstarter[0].EMmotorstarter[0].et200SpMotorstarterInputs[0..1].energySaving := FALSE;
   unitMotorstarter[0].EMmotorstarter[1].et200SpMotorstarterInputs[0..1].energySaving := FALSE;
   unitMotorstarter[0].EMmotorstarter[2].et200SpMotorstarterInputs[0..1].energySaving := FALSE;
   unitMotorstarter[0].EMmotorstarter[3].et200SpMotorstarterInputs[0..1].energySaving := FALSE;
   unitMotorstarter[0].EMmotorstarter[4].et200SpMotorstarterInputs[0..1].energySaving := FALSE;
   unitMotorstarter[0].EMmotorstarter[5].et200SpMotorstarterInputs[0..1].energySaving := FALSE;
   unitMotorstarter[0].EMmotorstarter[6].et200SpMotorstarterInputs[0..1].energySaving := FALSE;
   unitMotorstarter[0].EMmotorstarter[7].et200SpMotorstarterInputs[0..1].energySaving := FALSE;
   unitMotorstarter[0].EMmotorstarter[0].et200SpMotorstarterInputs[0..1].moduleInserted := FALSE;
   unitMotorstarter[0].EMmotorstarter[1].et200SpMotorstarterInputs[0..1].moduleInserted := FALSE;
   unitMotorstarter[0].EMmotorstarter[2].et200SpMotorstarterInputs[0..1].moduleInserted := FALSE;
   unitMotorstarter[0].EMmotorstarter[3].et200SpMotorstarterInputs[0..1].moduleInserted := FALSE;
   unitMotorstarter[0].EMmotorstarter[4].et200SpMotorstarterInputs[0..1].moduleInserted := FALSE;
   unitMotorstarter[0].EMmotorstarter[5].et200SpMotorstarterInputs[0..1].moduleInserted := FALSE;
   unitMotorstarter[0].EMmotorstarter[6].et200SpMotorstarterInputs[0..1].moduleInserted := FALSE;
   unitMotorstarter[0].EMmotorstarter[7].et200SpMotorstarterInputs[0..1].moduleInserted := FALSE;
   unitMotorstarter[0].EMmotorstarter[0].et200SpMotorstarterInputs[0..1].exProtectionMotorActive := FALSE;
   unitMotorstarter[0].EMmotorstarter[1].et200SpMotorstarterInputs[0..1].exProtectionMotorActive := FALSE;
   unitMotorstarter[0].EMmotorstarter[2].et200SpMotorstarterInputs[0..1].exProtectionMotorActive := FALSE;
   unitMotorstarter[0].EMmotorstarter[3].et200SpMotorstarterInputs[0..1].exProtectionMotorActive := FALSE;
   unitMotorstarter[0].EMmotorstarter[4].et200SpMotorstarterInputs[0..1].exProtectionMotorActive := FALSE;
   unitMotorstarter[0].EMmotorstarter[5].et200SpMotorstarterInputs[0..1].exProtectionMotorActive := FALSE;
   unitMotorstarter[0].EMmotorstarter[6].et200SpMotorstarterInputs[0..1].exProtectionMotorActive := FALSE;
   unitMotorstarter[0].EMmotorstarter[7].et200SpMotorstarterInputs[0..1].exProtectionMotorActive := FALSE;
   unitMotorstarter[0].EMmotorstarter[0].et200SpMotorstarterInputs[0..1].blockActive := FALSE;
   unitMotorstarter[0].EMmotorstarter[1].et200SpMotorstarterInputs[0..1].blockActive := FALSE;
   unitMotorstarter[0].EMmotorstarter[2].et200SpMotorstarterInputs[0..1].blockActive := FALSE;
   unitMotorstarter[0].EMmotorstarter[3].et200SpMotorstarterInputs[0..1].blockActive := FALSE;
   unitMotorstarter[0].EMmotorstarter[4].et200SpMotorstarterInputs[0..1].blockActive := FALSE;
   unitMotorstarter[0].EMmotorstarter[5].et200SpMotorstarterInputs[0..1].blockActive := FALSE;
   unitMotorstarter[0].EMmotorstarter[6].et200SpMotorstarterInputs[0..1].blockActive := FALSE;
   unitMotorstarter[0].EMmotorstarter[7].et200SpMotorstarterInputs[0..1].blockActive := FALSE;
   unitMotorstarter[0].EMmotorstarter[0].et200SpMotorstarterInputs[0..1].thermalMotorOverload := FALSE;
   unitMotorstarter[0].EMmotorstarter[1].et200SpMotorstarterInputs[0..1].thermalMotorOverload := FALSE;
   unitMotorstarter[0].EMmotorstarter[2].et200SpMotorstarterInputs[0..1].thermalMotorOverload := FALSE;
   unitMotorstarter[0].EMmotorstarter[3].et200SpMotorstarterInputs[0..1].thermalMotorOverload := FALSE;
   unitMotorstarter[0].EMmotorstarter[4].et200SpMotorstarterInputs[0..1].thermalMotorOverload := FALSE;
   unitMotorstarter[0].EMmotorstarter[5].et200SpMotorstarterInputs[0..1].thermalMotorOverload := FALSE;
   unitMotorstarter[0].EMmotorstarter[6].et200SpMotorstarterInputs[0..1].thermalMotorOverload := FALSE;
   unitMotorstarter[0].EMmotorstarter[7].et200SpMotorstarterInputs[0..1].thermalMotorOverload := FALSE;
   unitMotorstarter[0].EMmotorstarter[0].et200SpMotorstarterInputs[0..1].spare5 := FALSE;
   unitMotorstarter[0].EMmotorstarter[1].et200SpMotorstarterInputs[0..1].spare5 := FALSE;
   unitMotorstarter[0].EMmotorstarter[2].et200SpMotorstarterInputs[0..1].spare5 := FALSE;
   unitMotorstarter[0].EMmotorstarter[3].et200SpMotorstarterInputs[0..1].spare5 := FALSE;
   unitMotorstarter[0].EMmotorstarter[4].et200SpMotorstarterInputs[0..1].spare5 := FALSE;
   unitMotorstarter[0].EMmotorstarter[5].et200SpMotorstarterInputs[0..1].spare5 := FALSE;
   unitMotorstarter[0].EMmotorstarter[6].et200SpMotorstarterInputs[0..1].spare5 := FALSE;
   unitMotorstarter[0].EMmotorstarter[7].et200SpMotorstarterInputs[0..1].spare5 := FALSE;
   unitMotorstarter[0].EMmotorstarter[0].et200SpMotorstarterInputs[0..1].currentLimitTripping := FALSE;
   unitMotorstarter[0].EMmotorstarter[1].et200SpMotorstarterInputs[0..1].currentLimitTripping := FALSE;
   unitMotorstarter[0].EMmotorstarter[2].et200SpMotorstarterInputs[0..1].currentLimitTripping := FALSE;
   unitMotorstarter[0].EMmotorstarter[3].et200SpMotorstarterInputs[0..1].currentLimitTripping := FALSE;
   unitMotorstarter[0].EMmotorstarter[4].et200SpMotorstarterInputs[0..1].currentLimitTripping := FALSE;
   unitMotorstarter[0].EMmotorstarter[5].et200SpMotorstarterInputs[0..1].currentLimitTripping := FALSE;
   unitMotorstarter[0].EMmotorstarter[6].et200SpMotorstarterInputs[0..1].currentLimitTripping := FALSE;
   unitMotorstarter[0].EMmotorstarter[7].et200SpMotorstarterInputs[0..1].currentLimitTripping := FALSE;
   unitMotorstarter[0].EMmotorstarter[0].et200SpMotorstarterInputs[0..1].statusFailDi := FALSE;
   unitMotorstarter[0].EMmotorstarter[1].et200SpMotorstarterInputs[0..1].statusFailDi := FALSE;
   unitMotorstarter[0].EMmotorstarter[2].et200SpMotorstarterInputs[0..1].statusFailDi := FALSE;
   unitMotorstarter[0].EMmotorstarter[3].et200SpMotorstarterInputs[0..1].statusFailDi := FALSE;
   unitMotorstarter[0].EMmotorstarter[4].et200SpMotorstarterInputs[0..1].statusFailDi := FALSE;
   unitMotorstarter[0].EMmotorstarter[5].et200SpMotorstarterInputs[0..1].statusFailDi := FALSE;
   unitMotorstarter[0].EMmotorstarter[6].et200SpMotorstarterInputs[0..1].statusFailDi := FALSE;
   unitMotorstarter[0].EMmotorstarter[7].et200SpMotorstarterInputs[0..1].statusFailDi := FALSE;
   unitMotorstarter[0].EMmotorstarter[0].et200SpMotorstarterInputs[0..1].residualCurrent := FALSE;
   unitMotorstarter[0].EMmotorstarter[1].et200SpMotorstarterInputs[0..1].residualCurrent := FALSE;
   unitMotorstarter[0].EMmotorstarter[2].et200SpMotorstarterInputs[0..1].residualCurrent := FALSE;
   unitMotorstarter[0].EMmotorstarter[3].et200SpMotorstarterInputs[0..1].residualCurrent := FALSE;
   unitMotorstarter[0].EMmotorstarter[4].et200SpMotorstarterInputs[0..1].residualCurrent := FALSE;
   unitMotorstarter[0].EMmotorstarter[5].et200SpMotorstarterInputs[0..1].residualCurrent := FALSE;
   unitMotorstarter[0].EMmotorstarter[6].et200SpMotorstarterInputs[0..1].residualCurrent := FALSE;
   unitMotorstarter[0].EMmotorstarter[7].et200SpMotorstarterInputs[0..1].residualCurrent := FALSE;
   unitMotorstarter[0].EMmotorstarter[0].et200SpMotorstarterInputs[0..1].asymmetryDetected := FALSE;
   unitMotorstarter[0].EMmotorstarter[1].et200SpMotorstarterInputs[0..1].asymmetryDetected := FALSE;
   unitMotorstarter[0].EMmotorstarter[2].et200SpMotorstarterInputs[0..1].asymmetryDetected := FALSE;
   unitMotorstarter[0].EMmotorstarter[3].et200SpMotorstarterInputs[0..1].asymmetryDetected := FALSE;
   unitMotorstarter[0].EMmotorstarter[4].et200SpMotorstarterInputs[0..1].asymmetryDetected := FALSE;
   unitMotorstarter[0].EMmotorstarter[5].et200SpMotorstarterInputs[0..1].asymmetryDetected := FALSE;
   unitMotorstarter[0].EMmotorstarter[6].et200SpMotorstarterInputs[0..1].asymmetryDetected := FALSE;
   unitMotorstarter[0].EMmotorstarter[7].et200SpMotorstarterInputs[0..1].asymmetryDetected := FALSE;
   unitMotorstarter[0].EMmotorstarter[0].et200SpMotorstarterInputs[0..1].overtemperature := FALSE;
   unitMotorstarter[0].EMmotorstarter[1].et200SpMotorstarterInputs[0..1].overtemperature := FALSE;
   unitMotorstarter[0].EMmotorstarter[2].et200SpMotorstarterInputs[0..1].overtemperature := FALSE;
   unitMotorstarter[0].EMmotorstarter[3].et200SpMotorstarterInputs[0..1].overtemperature := FALSE;
   unitMotorstarter[0].EMmotorstarter[4].et200SpMotorstarterInputs[0..1].overtemperature := FALSE;
   unitMotorstarter[0].EMmotorstarter[5].et200SpMotorstarterInputs[0..1].overtemperature := FALSE;
   unitMotorstarter[0].EMmotorstarter[6].et200SpMotorstarterInputs[0..1].overtemperature := FALSE;
   unitMotorstarter[0].EMmotorstarter[7].et200SpMotorstarterInputs[0..1].overtemperature := FALSE;
   unitMotorstarter[0].EMmotorstarter[0].et200SpMotorstarterInputs[0..1].spare7 := FALSE;
   unitMotorstarter[0].EMmotorstarter[1].et200SpMotorstarterInputs[0..1].spare7 := FALSE;
   unitMotorstarter[0].EMmotorstarter[2].et200SpMotorstarterInputs[0..1].spare7 := FALSE;
   unitMotorstarter[0].EMmotorstarter[3].et200SpMotorstarterInputs[0..1].spare7 := FALSE;
   unitMotorstarter[0].EMmotorstarter[4].et200SpMotorstarterInputs[0..1].spare7 := FALSE;
   unitMotorstarter[0].EMmotorstarter[5].et200SpMotorstarterInputs[0..1].spare7 := FALSE;
   unitMotorstarter[0].EMmotorstarter[6].et200SpMotorstarterInputs[0..1].spare7 := FALSE;
   unitMotorstarter[0].EMmotorstarter[7].et200SpMotorstarterInputs[0..1].spare7 := FALSE;
   unitMotorstarter[0].EMmotorstarter[0].et200SpMotorstarterOutputs[0..1].motorCw := FALSE;
   unitMotorstarter[0].EMmotorstarter[1].et200SpMotorstarterOutputs[0..1].motorCw := FALSE;
   unitMotorstarter[0].EMmotorstarter[2].et200SpMotorstarterOutputs[0..1].motorCw := FALSE;
   unitMotorstarter[0].EMmotorstarter[3].et200SpMotorstarterOutputs[0..1].motorCw := FALSE;
   unitMotorstarter[0].EMmotorstarter[4].et200SpMotorstarterOutputs[0..1].motorCw := FALSE;
   unitMotorstarter[0].EMmotorstarter[5].et200SpMotorstarterOutputs[0..1].motorCw := FALSE;
   unitMotorstarter[0].EMmotorstarter[6].et200SpMotorstarterOutputs[0..1].motorCw := FALSE;
   unitMotorstarter[0].EMmotorstarter[7].et200SpMotorstarterOutputs[0..1].motorCw := FALSE;
   unitMotorstarter[0].EMmotorstarter[0].et200SpMotorstarterOutputs[0..1].motorCww := FALSE;
   unitMotorstarter[0].EMmotorstarter[1].et200SpMotorstarterOutputs[0..1].motorCww := FALSE;
   unitMotorstarter[0].EMmotorstarter[2].et200SpMotorstarterOutputs[0..1].motorCww := FALSE;
   unitMotorstarter[0].EMmotorstarter[3].et200SpMotorstarterOutputs[0..1].motorCww := FALSE;
   unitMotorstarter[0].EMmotorstarter[4].et200SpMotorstarterOutputs[0..1].motorCww := FALSE;
   unitMotorstarter[0].EMmotorstarter[5].et200SpMotorstarterOutputs[0..1].motorCww := FALSE;
   unitMotorstarter[0].EMmotorstarter[6].et200SpMotorstarterOutputs[0..1].motorCww := FALSE;
   unitMotorstarter[0].EMmotorstarter[7].et200SpMotorstarterOutputs[0..1].motorCww := FALSE;
   unitMotorstarter[0].EMmotorstarter[0].et200SpMotorstarterOutputs[0..1].reserve1 := FALSE;
   unitMotorstarter[0].EMmotorstarter[1].et200SpMotorstarterOutputs[0..1].reserve1 := FALSE;
   unitMotorstarter[0].EMmotorstarter[2].et200SpMotorstarterOutputs[0..1].reserve1 := FALSE;
   unitMotorstarter[0].EMmotorstarter[3].et200SpMotorstarterOutputs[0..1].reserve1 := FALSE;
   unitMotorstarter[0].EMmotorstarter[4].et200SpMotorstarterOutputs[0..1].reserve1 := FALSE;
   unitMotorstarter[0].EMmotorstarter[5].et200SpMotorstarterOutputs[0..1].reserve1 := FALSE;
   unitMotorstarter[0].EMmotorstarter[6].et200SpMotorstarterOutputs[0..1].reserve1 := FALSE;
   unitMotorstarter[0].EMmotorstarter[7].et200SpMotorstarterOutputs[0..1].reserve1 := FALSE;
   unitMotorstarter[0].EMmotorstarter[0].et200SpMotorstarterOutputs[0..1].tripReset := FALSE;
   unitMotorstarter[0].EMmotorstarter[1].et200SpMotorstarterOutputs[0..1].tripReset := FALSE;
   unitMotorstarter[0].EMmotorstarter[2].et200SpMotorstarterOutputs[0..1].tripReset := FALSE;
   unitMotorstarter[0].EMmotorstarter[3].et200SpMotorstarterOutputs[0..1].tripReset := FALSE;
   unitMotorstarter[0].EMmotorstarter[4].et200SpMotorstarterOutputs[0..1].tripReset := FALSE;
   unitMotorstarter[0].EMmotorstarter[5].et200SpMotorstarterOutputs[0..1].tripReset := FALSE;
   unitMotorstarter[0].EMmotorstarter[6].et200SpMotorstarterOutputs[0..1].tripReset := FALSE;
   unitMotorstarter[0].EMmotorstarter[7].et200SpMotorstarterOutputs[0..1].tripReset := FALSE;
   unitMotorstarter[0].EMmotorstarter[0].et200SpMotorstarterOutputs[0..1].emergencyStart := FALSE;
   unitMotorstarter[0].EMmotorstarter[1].et200SpMotorstarterOutputs[0..1].emergencyStart := FALSE;
   unitMotorstarter[0].EMmotorstarter[2].et200SpMotorstarterOutputs[0..1].emergencyStart := FALSE;
   unitMotorstarter[0].EMmotorstarter[3].et200SpMotorstarterOutputs[0..1].emergencyStart := FALSE;
   unitMotorstarter[0].EMmotorstarter[4].et200SpMotorstarterOutputs[0..1].emergencyStart := FALSE;
   unitMotorstarter[0].EMmotorstarter[5].et200SpMotorstarterOutputs[0..1].emergencyStart := FALSE;
   unitMotorstarter[0].EMmotorstarter[6].et200SpMotorstarterOutputs[0..1].emergencyStart := FALSE;
   unitMotorstarter[0].EMmotorstarter[7].et200SpMotorstarterOutputs[0..1].emergencyStart := FALSE;
   unitMotorstarter[0].EMmotorstarter[0].et200SpMotorstarterOutputs[0..1].reserve2 := FALSE;
   unitMotorstarter[0].EMmotorstarter[1].et200SpMotorstarterOutputs[0..1].reserve2 := FALSE;
   unitMotorstarter[0].EMmotorstarter[2].et200SpMotorstarterOutputs[0..1].reserve2 := FALSE;
   unitMotorstarter[0].EMmotorstarter[3].et200SpMotorstarterOutputs[0..1].reserve2 := FALSE;
   unitMotorstarter[0].EMmotorstarter[4].et200SpMotorstarterOutputs[0..1].reserve2 := FALSE;
   unitMotorstarter[0].EMmotorstarter[5].et200SpMotorstarterOutputs[0..1].reserve2 := FALSE;
   unitMotorstarter[0].EMmotorstarter[6].et200SpMotorstarterOutputs[0..1].reserve2 := FALSE;
   unitMotorstarter[0].EMmotorstarter[7].et200SpMotorstarterOutputs[0..1].reserve2 := FALSE;
   unitMotorstarter[0].EMmotorstarter[0].et200SpMotorstarterOutputs[0..1].reserve3 := FALSE;
   unitMotorstarter[0].EMmotorstarter[1].et200SpMotorstarterOutputs[0..1].reserve3 := FALSE;
   unitMotorstarter[0].EMmotorstarter[2].et200SpMotorstarterOutputs[0..1].reserve3 := FALSE;
   unitMotorstarter[0].EMmotorstarter[3].et200SpMotorstarterOutputs[0..1].reserve3 := FALSE;
   unitMotorstarter[0].EMmotorstarter[4].et200SpMotorstarterOutputs[0..1].reserve3 := FALSE;
   unitMotorstarter[0].EMmotorstarter[5].et200SpMotorstarterOutputs[0..1].reserve3 := FALSE;
   unitMotorstarter[0].EMmotorstarter[6].et200SpMotorstarterOutputs[0..1].reserve3 := FALSE;
   unitMotorstarter[0].EMmotorstarter[7].et200SpMotorstarterOutputs[0..1].reserve3 := FALSE;
   unitMotorstarter[0].EMmotorstarter[0].et200SpMotorstarterOutputs[0..1].coldStart := FALSE;
   unitMotorstarter[0].EMmotorstarter[1].et200SpMotorstarterOutputs[0..1].coldStart := FALSE;
   unitMotorstarter[0].EMmotorstarter[2].et200SpMotorstarterOutputs[0..1].coldStart := FALSE;
   unitMotorstarter[0].EMmotorstarter[3].et200SpMotorstarterOutputs[0..1].coldStart := FALSE;
   unitMotorstarter[0].EMmotorstarter[4].et200SpMotorstarterOutputs[0..1].coldStart := FALSE;
   unitMotorstarter[0].EMmotorstarter[5].et200SpMotorstarterOutputs[0..1].coldStart := FALSE;
   unitMotorstarter[0].EMmotorstarter[6].et200SpMotorstarterOutputs[0..1].coldStart := FALSE;
   unitMotorstarter[0].EMmotorstarter[7].et200SpMotorstarterOutputs[0..1].coldStart := FALSE;
   unitMotorstarter[0].EMmotorstarter[0].et200SpMotorstarterOutputs[0..1].reserve4 := FALSE;
   unitMotorstarter[0].EMmotorstarter[1].et200SpMotorstarterOutputs[0..1].reserve4 := FALSE;
   unitMotorstarter[0].EMmotorstarter[2].et200SpMotorstarterOutputs[0..1].reserve4 := FALSE;
   unitMotorstarter[0].EMmotorstarter[3].et200SpMotorstarterOutputs[0..1].reserve4 := FALSE;
   unitMotorstarter[0].EMmotorstarter[4].et200SpMotorstarterOutputs[0..1].reserve4 := FALSE;
   unitMotorstarter[0].EMmotorstarter[5].et200SpMotorstarterOutputs[0..1].reserve4 := FALSE;
   unitMotorstarter[0].EMmotorstarter[6].et200SpMotorstarterOutputs[0..1].reserve4 := FALSE;
   unitMotorstarter[0].EMmotorstarter[7].et200SpMotorstarterOutputs[0..1].reserve4 := FALSE;
   unitMotorstarter[0].EMmotorstarter[0].et200SpMotorstarterOutputs[0..1].reserve5 := FALSE;
   unitMotorstarter[0].EMmotorstarter[1].et200SpMotorstarterOutputs[0..1].reserve5 := FALSE;
   unitMotorstarter[0].EMmotorstarter[2].et200SpMotorstarterOutputs[0..1].reserve5 := FALSE;
   unitMotorstarter[0].EMmotorstarter[3].et200SpMotorstarterOutputs[0..1].reserve5 := FALSE;
   unitMotorstarter[0].EMmotorstarter[4].et200SpMotorstarterOutputs[0..1].reserve5 := FALSE;
   unitMotorstarter[0].EMmotorstarter[5].et200SpMotorstarterOutputs[0..1].reserve5 := FALSE;
   unitMotorstarter[0].EMmotorstarter[6].et200SpMotorstarterOutputs[0..1].reserve5 := FALSE;
   unitMotorstarter[0].EMmotorstarter[7].et200SpMotorstarterOutputs[0..1].reserve5 := FALSE;
   unitMotorstarter[0].EMmotorstarter[0].et200SpMotorstarterOutputs[0..1].reserve6 := FALSE;
   unitMotorstarter[0].EMmotorstarter[1].et200SpMotorstarterOutputs[0..1].reserve6 := FALSE;
   unitMotorstarter[0].EMmotorstarter[2].et200SpMotorstarterOutputs[0..1].reserve6 := FALSE;
   unitMotorstarter[0].EMmotorstarter[3].et200SpMotorstarterOutputs[0..1].reserve6 := FALSE;
   unitMotorstarter[0].EMmotorstarter[4].et200SpMotorstarterOutputs[0..1].reserve6 := FALSE;
   unitMotorstarter[0].EMmotorstarter[5].et200SpMotorstarterOutputs[0..1].reserve6 := FALSE;
   unitMotorstarter[0].EMmotorstarter[6].et200SpMotorstarterOutputs[0..1].reserve6 := FALSE;
   unitMotorstarter[0].EMmotorstarter[7].et200SpMotorstarterOutputs[0..1].reserve6 := FALSE;
   unitMotorstarter[0].EMmotorstarter[0].et200SpMotorstarterOutputs[0..1].reserve7 := FALSE;
   unitMotorstarter[0].EMmotorstarter[1].et200SpMotorstarterOutputs[0..1].reserve7 := FALSE;
   unitMotorstarter[0].EMmotorstarter[2].et200SpMotorstarterOutputs[0..1].reserve7 := FALSE;
   unitMotorstarter[0].EMmotorstarter[3].et200SpMotorstarterOutputs[0..1].reserve7 := FALSE;
   unitMotorstarter[0].EMmotorstarter[4].et200SpMotorstarterOutputs[0..1].reserve7 := FALSE;
   unitMotorstarter[0].EMmotorstarter[5].et200SpMotorstarterOutputs[0..1].reserve7 := FALSE;
   unitMotorstarter[0].EMmotorstarter[6].et200SpMotorstarterOutputs[0..1].reserve7 := FALSE;
   unitMotorstarter[0].EMmotorstarter[7].et200SpMotorstarterOutputs[0..1].reserve7 := FALSE;
   unitMotorstarter[0].EMmotorstarter[0].et200SpMotorstarterOutputs[0..1].reserve8 := FALSE;
   unitMotorstarter[0].EMmotorstarter[1].et200SpMotorstarterOutputs[0..1].reserve8 := FALSE;
   unitMotorstarter[0].EMmotorstarter[2].et200SpMotorstarterOutputs[0..1].reserve8 := FALSE;
   unitMotorstarter[0].EMmotorstarter[3].et200SpMotorstarterOutputs[0..1].reserve8 := FALSE;
   unitMotorstarter[0].EMmotorstarter[4].et200SpMotorstarterOutputs[0..1].reserve8 := FALSE;
   unitMotorstarter[0].EMmotorstarter[5].et200SpMotorstarterOutputs[0..1].reserve8 := FALSE;
   unitMotorstarter[0].EMmotorstarter[6].et200SpMotorstarterOutputs[0..1].reserve8 := FALSE;
   unitMotorstarter[0].EMmotorstarter[7].et200SpMotorstarterOutputs[0..1].reserve8 := FALSE;
   unitMotorstarter[0].EMmotorstarter[0].et200SpMotorstarterOutputs[0..1].reserve9 := FALSE;
   unitMotorstarter[0].EMmotorstarter[1].et200SpMotorstarterOutputs[0..1].reserve9 := FALSE;
   unitMotorstarter[0].EMmotorstarter[2].et200SpMotorstarterOutputs[0..1].reserve9 := FALSE;
   unitMotorstarter[0].EMmotorstarter[3].et200SpMotorstarterOutputs[0..1].reserve9 := FALSE;
   unitMotorstarter[0].EMmotorstarter[4].et200SpMotorstarterOutputs[0..1].reserve9 := FALSE;
   unitMotorstarter[0].EMmotorstarter[5].et200SpMotorstarterOutputs[0..1].reserve9 := FALSE;
   unitMotorstarter[0].EMmotorstarter[6].et200SpMotorstarterOutputs[0..1].reserve9 := FALSE;
   unitMotorstarter[0].EMmotorstarter[7].et200SpMotorstarterOutputs[0..1].reserve9 := FALSE;
   unitMotorstarter[0].EMmotorstarter[0].et200SpMotorstarterOutputs[0..1].reserve10 := FALSE;
   unitMotorstarter[0].EMmotorstarter[1].et200SpMotorstarterOutputs[0..1].reserve10 := FALSE;
   unitMotorstarter[0].EMmotorstarter[2].et200SpMotorstarterOutputs[0..1].reserve10 := FALSE;
   unitMotorstarter[0].EMmotorstarter[3].et200SpMotorstarterOutputs[0..1].reserve10 := FALSE;
   unitMotorstarter[0].EMmotorstarter[4].et200SpMotorstarterOutputs[0..1].reserve10 := FALSE;
   unitMotorstarter[0].EMmotorstarter[5].et200SpMotorstarterOutputs[0..1].reserve10 := FALSE;
   unitMotorstarter[0].EMmotorstarter[6].et200SpMotorstarterOutputs[0..1].reserve10 := FALSE;
   unitMotorstarter[0].EMmotorstarter[7].et200SpMotorstarterOutputs[0..1].reserve10 := FALSE;
   unitMotorstarter[0].EMmotorstarter[0].et200SpMotorstarterOutputs[0..1].disableQuickStop := FALSE;
   unitMotorstarter[0].EMmotorstarter[1].et200SpMotorstarterOutputs[0..1].disableQuickStop := FALSE;
   unitMotorstarter[0].EMmotorstarter[2].et200SpMotorstarterOutputs[0..1].disableQuickStop := FALSE;
   unitMotorstarter[0].EMmotorstarter[3].et200SpMotorstarterOutputs[0..1].disableQuickStop := FALSE;
   unitMotorstarter[0].EMmotorstarter[4].et200SpMotorstarterOutputs[0..1].disableQuickStop := FALSE;
   unitMotorstarter[0].EMmotorstarter[5].et200SpMotorstarterOutputs[0..1].disableQuickStop := FALSE;
   unitMotorstarter[0].EMmotorstarter[6].et200SpMotorstarterOutputs[0..1].disableQuickStop := FALSE;
   unitMotorstarter[0].EMmotorstarter[7].et200SpMotorstarterOutputs[0..1].disableQuickStop := FALSE;
END_DATA_BLOCK

ORGANIZATION_BLOCK "Main"   // OB1, LAD, ProgramCycle
TITLE = "Main Program Sweep (Cycle)"
// stored: AutoNumber false, IsIECCheckEnabled true, SetENOAutomatically true
   VAR_INPUT
      Initial_Call : Bool;   // Initial call of this OB
      Remanence : Bool;   // =True, if remanent data are available
   END_VAR
   VAR_TEMP   // added for the SCL form of the ladder/FBD networks
      _w1 : Bool;
      _w2 : Bool;
      _w3 : Bool;
      _w4 : Bool;
      _w5 : Bool;
      _w6 : Bool;
   END_VAR
BEGIN

REGION Network 1: First Cycle
   // Set bit to true in first cycle, and false in all other cycles
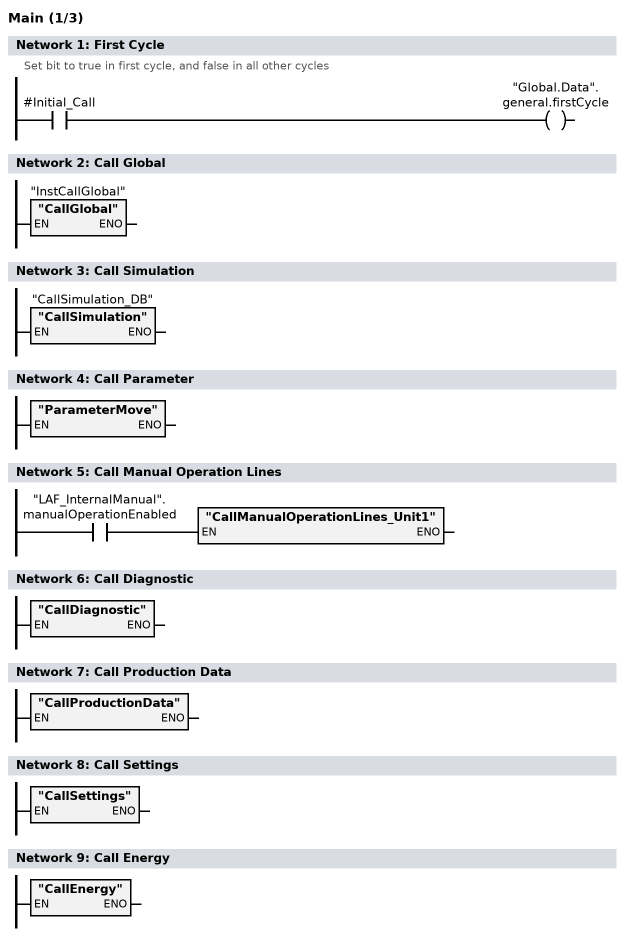
   RUNG wire#powerrail
      Contact( #Initial_Call )
      Coil( "Global.Data".general.firstCycle )
   END_RUNG
   // the same network as SCL:
   "Global.Data".general.firstCycle := #Initial_Call;
END_REGION

REGION Network 2: Call Global
   RUNG wire#powerrail
      "InstCallGlobal"()
   END_RUNG
   // the same network as SCL:
   "InstCallGlobal"();   // "CallGlobal"
END_REGION

REGION Network 3: Call Simulation
   RUNG wire#powerrail
      "CallSimulation_DB"()
   END_RUNG
   // the same network as SCL:
   "CallSimulation_DB"();   // "CallSimulation"
END_REGION

REGION Network 4: Call Parameter
   RUNG wire#powerrail
      "ParameterMove"()
   END_RUNG
   // the same network as SCL:
   "ParameterMove"();
END_REGION

REGION Network 5: Call Manual Operation Lines
   RUNG wire#powerrail
      Contact( "LAF_InternalManual".manualOperationEnabled )
      "CallManualOperationLines_Unit1"()
   END_RUNG
   // the same network as SCL:
   IF "LAF_InternalManual".manualOperationEnabled THEN "CallManualOperationLines_Unit1"(); END_IF;
END_REGION

REGION Network 6: Call Diagnostic
   RUNG wire#powerrail
      "CallDiagnostic"()
   END_RUNG
   // the same network as SCL:
   "CallDiagnostic"();
END_REGION

REGION Network 7: Call Production Data
   RUNG wire#powerrail
      "CallProductionData"()
   END_RUNG
   // the same network as SCL:
   "CallProductionData"();
END_REGION

REGION Network 8: Call Settings
   RUNG wire#powerrail
      "CallSettings"()
   END_RUNG
   // the same network as SCL:
   "CallSettings"();
END_REGION

REGION Network 9: Call Energy
   RUNG wire#powerrail
      "CallEnergy"()
   END_RUNG
   // the same network as SCL:
   "CallEnergy"();
END_REGION

